Yaskawa INFORM job: DEMO_ROOF_UPPER_0625_3PAINT_5.JBI

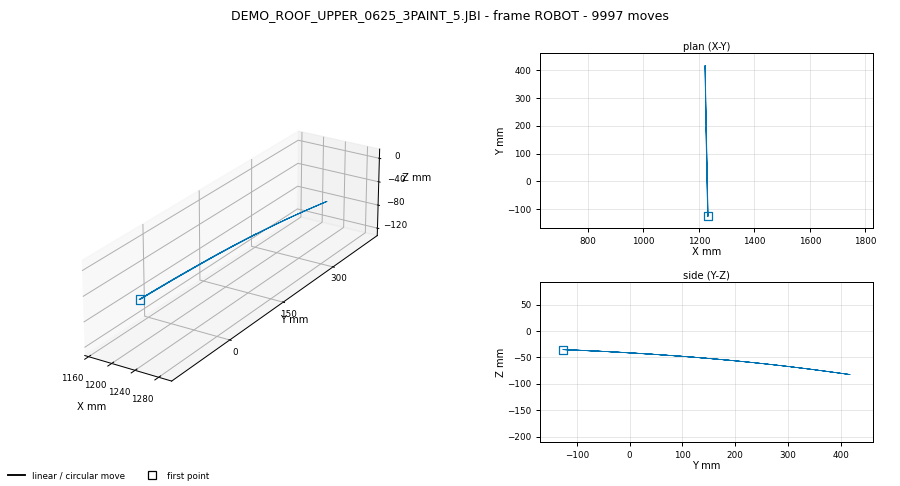
[picture p0: tool path of DEMO_ROOF_UPPER_0625_3PAINT_5.JBI in frame ROBOT, 9997 of 9997 moves have a stored position in this frame; points joined in program order, loops and branches not executed]
/JOB
//NAME DEMO_ROOF_UPPER_0625_3PAINT5
//POS
///NPOS 9997,0,0,0,0,0
///TOOL 0
///USER 0
///POSTYPE ROBOT
///RECTAN
///RCONF 1,0,0,0,0,0,0,0,0,0,0,0,0,0,0,0,0,0,0,0,0,0,0,0
C00000=1233.237,-125.531,-35.008,179.340,5.259,149.111
C00001=1233.231,-125.281,-35.017,179.342,5.259,149.110
C00002=1233.226,-125.032,-35.027,179.345,5.260,149.110
C00003=1233.220,-124.782,-35.037,179.347,5.259,149.109
C00004=1233.215,-124.532,-35.046,179.350,5.260,149.108
C00005=1233.210,-124.282,-35.057,179.352,5.259,149.107
C00006=1233.205,-124.033,-35.067,179.354,5.260,149.107
C00007=1233.199,-123.783,-35.076,179.356,5.260,149.106
C00008=1233.194,-123.533,-35.086,179.359,5.260,149.105
C00009=1233.189,-123.284,-35.096,179.361,5.260,149.105
C00010=1233.184,-123.033,-35.105,179.363,5.259,149.104
C00011=1233.178,-122.784,-35.116,179.366,5.260,149.103
C00012=1233.173,-122.534,-35.125,179.368,5.259,149.103
C00013=1233.168,-122.285,-35.136,179.370,5.260,149.102
C00014=1233.163,-122.034,-35.145,179.372,5.260,149.101
C00015=1233.157,-121.785,-35.155,179.375,5.260,149.101
C00016=1233.152,-121.535,-35.165,179.377,5.260,149.100
C00017=1233.147,-121.286,-35.175,179.379,5.260,149.099
C00018=1233.142,-121.035,-35.185,179.381,5.260,149.099
C00019=1233.136,-120.786,-35.195,179.384,5.260,149.098
C00020=1233.131,-120.536,-35.205,179.386,5.260,149.097
C00021=1233.126,-120.287,-35.215,179.388,5.260,149.096
C00022=1233.121,-120.037,-35.225,179.391,5.260,149.096
C00023=1233.115,-119.787,-35.234,179.393,5.260,149.095
C00024=1233.110,-119.537,-35.244,179.395,5.260,149.094
C00025=1233.105,-119.288,-35.254,179.397,5.260,149.094
C00026=1233.100,-119.038,-35.265,179.400,5.261,149.093
C00027=1233.094,-118.788,-35.275,179.402,5.260,149.092
C00028=1233.089,-118.539,-35.285,179.404,5.260,149.092
C00029=1233.084,-118.288,-35.294,179.407,5.260,149.091
C00030=1233.079,-118.038,-35.304,179.409,5.260,149.090
C00031=1233.073,-117.789,-35.315,179.412,5.260,149.089
C00032=1233.069,-117.539,-35.325,179.414,5.260,149.089
C00033=1233.063,-117.289,-35.335,179.416,5.261,149.088
C00034=1233.058,-117.040,-35.345,179.418,5.260,149.088
C00035=1233.053,-116.791,-35.355,179.421,5.261,149.087
C00036=1233.048,-116.540,-35.365,179.423,5.260,149.086
C00037=1233.042,-116.290,-35.375,179.426,5.261,149.085
C00038=1233.036,-116.041,-35.385,179.428,5.260,149.085
C00039=1233.032,-115.791,-35.395,179.430,5.260,149.084
C00040=1233.026,-115.541,-35.405,179.432,5.261,149.083
C00041=1233.021,-115.292,-35.415,179.435,5.260,149.083
C00042=1233.016,-115.041,-35.426,179.437,5.261,149.082
C00043=1233.011,-114.792,-35.436,179.439,5.260,149.081
C00044=1233.005,-114.543,-35.446,179.441,5.261,149.081
C00045=1233.000,-114.292,-35.456,179.444,5.261,149.080
C00046=1232.995,-114.043,-35.467,179.446,5.261,149.079
C00047=1232.990,-113.794,-35.476,179.448,5.261,149.078
C00048=1232.985,-113.543,-35.487,179.450,5.260,149.078
C00049=1232.979,-113.294,-35.497,179.453,5.261,149.077
C00050=1232.974,-113.044,-35.507,179.455,5.260,149.076
C00051=1232.969,-112.794,-35.518,179.458,5.261,149.076
C00052=1232.964,-112.545,-35.527,179.460,5.260,149.075
C00053=1232.959,-112.295,-35.538,179.463,5.261,149.074
C00054=1232.953,-112.045,-35.548,179.465,5.261,149.073
C00055=1232.948,-111.796,-35.558,179.467,5.261,149.073
C00056=1232.943,-111.545,-35.569,179.470,5.261,149.072
C00057=1232.938,-111.296,-35.579,179.472,5.261,149.072
C00058=1232.932,-111.047,-35.589,179.474,5.261,149.071
C00059=1232.927,-110.796,-35.599,179.476,5.261,149.070
C00060=1232.921,-110.547,-35.610,179.479,5.261,149.069
C00061=1232.916,-110.296,-35.620,179.481,5.261,149.069
C00062=1232.911,-110.047,-35.630,179.483,5.261,149.068
C00063=1232.905,-109.797,-35.641,179.485,5.261,149.067
C00064=1232.901,-109.547,-35.650,179.488,5.261,149.067
C00065=1232.895,-109.298,-35.661,179.490,5.261,149.066
C00066=1232.891,-109.048,-35.672,179.493,5.261,149.065
C00067=1232.885,-108.799,-35.682,179.495,5.261,149.064
C00068=1232.880,-108.549,-35.692,179.498,5.261,149.064
C00069=1232.875,-108.299,-35.703,179.500,5.261,149.063
C00070=1232.869,-108.049,-35.713,179.502,5.261,149.062
C00071=1232.864,-107.799,-35.724,179.504,5.262,149.062
C00072=1232.859,-107.550,-35.733,179.506,5.261,149.061
C00073=1232.854,-107.300,-35.744,179.509,5.262,149.060
C00074=1232.849,-107.051,-35.755,179.511,5.261,149.060
C00075=1232.843,-106.801,-35.765,179.514,5.262,149.059
C00076=1232.838,-106.551,-35.776,179.516,5.261,149.058
C00077=1232.833,-106.301,-35.786,179.518,5.262,149.057
C00078=1232.828,-106.051,-35.796,179.520,5.261,149.057
C00079=1232.822,-105.802,-35.807,179.523,5.262,149.056
C00080=1232.817,-105.552,-35.818,179.525,5.261,149.055
C00081=1232.812,-105.302,-35.828,179.528,5.262,149.055
C00082=1232.807,-105.052,-35.839,179.530,5.262,149.054
C00083=1232.801,-104.803,-35.849,179.533,5.262,149.053
C00084=1232.796,-104.552,-35.859,179.535,5.262,149.052
C00085=1232.792,-104.304,-35.870,179.537,5.261,149.052
C00086=1232.787,-104.054,-35.880,179.540,5.262,149.051
C00087=1232.781,-103.804,-35.891,179.542,5.261,149.050
C00088=1232.776,-103.554,-35.901,179.544,5.262,149.050
C00089=1232.771,-103.305,-35.912,179.546,5.262,149.049
C00090=1232.765,-103.055,-35.922,179.549,5.262,149.048
C00091=1232.760,-102.805,-35.933,179.551,5.262,149.048
C00092=1232.755,-102.556,-35.943,179.553,5.262,149.047
C00093=1232.750,-102.306,-35.954,179.555,5.262,149.046
C00094=1232.745,-102.056,-35.965,179.558,5.262,149.046
C00095=1232.739,-101.806,-35.975,179.560,5.262,149.045
C00096=1232.735,-101.556,-35.986,179.563,5.262,149.044
C00097=1232.729,-101.307,-35.997,179.565,5.262,149.043
C00098=1232.724,-101.057,-36.007,179.568,5.263,149.043
C00099=1232.718,-100.786,-36.019,179.570,5.262,149.042
C00100=1232.712,-100.515,-36.031,179.572,5.263,149.041
C00101=1232.707,-100.244,-36.042,179.575,5.262,149.040
C00102=1232.700,-99.973,-36.053,179.578,5.262,149.040
C00103=1232.696,-99.724,-36.065,179.580,5.262,149.039
C00104=1232.690,-99.474,-36.075,179.582,5.262,149.038
C00105=1232.685,-99.224,-36.086,179.585,5.262,149.037
C00106=1232.680,-98.975,-36.096,179.587,5.263,149.037
C00107=1232.675,-98.725,-36.107,179.589,5.262,149.036
C00108=1232.670,-98.475,-36.118,179.592,5.263,149.035
C00109=1232.665,-98.226,-36.129,179.594,5.262,149.035
C00110=1232.660,-97.975,-36.139,179.597,5.263,149.034
C00111=1232.654,-97.726,-36.150,179.599,5.262,149.033
C00112=1232.649,-97.476,-36.161,179.601,5.263,149.033
C00113=1232.644,-97.227,-36.172,179.603,5.263,149.032
C00114=1232.638,-96.977,-36.183,179.606,5.263,149.031
C00115=1232.633,-96.727,-36.193,179.608,5.263,149.031
C00116=1232.628,-96.477,-36.204,179.611,5.263,149.030
C00117=1232.623,-96.227,-36.215,179.613,5.263,149.029
C00118=1232.618,-95.978,-36.226,179.615,5.263,149.028
C00119=1232.613,-95.728,-36.236,179.617,5.263,149.028
C00120=1232.607,-95.479,-36.247,179.620,5.263,149.027
C00121=1232.602,-95.229,-36.258,179.622,5.263,149.026
C00122=1232.597,-94.979,-36.270,179.624,5.263,149.026
C00123=1232.591,-94.729,-36.280,179.627,5.263,149.025
C00124=1232.587,-94.480,-36.291,179.629,5.263,149.024
C00125=1232.581,-94.230,-36.301,179.632,5.263,149.023
C00126=1232.576,-93.981,-36.313,179.634,5.263,149.023
C00127=1232.571,-93.730,-36.323,179.637,5.263,149.022
C00128=1232.565,-93.481,-36.335,179.639,5.263,149.021
C00129=1232.560,-93.231,-36.345,179.641,5.264,149.021
C00130=1232.555,-92.982,-36.356,179.643,5.263,149.020
C00131=1232.550,-92.732,-36.367,179.646,5.264,149.019
C00132=1232.545,-92.482,-36.378,179.648,5.263,149.018
C00133=1232.539,-92.232,-36.389,179.651,5.264,149.018
C00134=1232.534,-91.983,-36.400,179.653,5.263,149.017
C00135=1232.529,-91.732,-36.411,179.656,5.264,149.016
C00136=1232.524,-91.483,-36.422,179.658,5.263,149.016
C00137=1232.519,-91.234,-36.433,179.660,5.264,149.015
C00138=1232.514,-90.983,-36.444,179.662,5.264,149.014
C00139=1232.508,-90.734,-36.455,179.665,5.264,149.013
C00140=1232.503,-90.484,-36.466,179.667,5.264,149.013
C00141=1232.499,-90.234,-36.477,179.670,5.264,149.012
C00142=1232.493,-89.985,-36.489,179.672,5.264,149.011
C00143=1232.488,-89.735,-36.499,179.675,5.264,149.011
C00144=1232.482,-89.486,-36.510,179.677,5.264,149.010
C00145=1232.477,-89.236,-36.521,179.679,5.264,149.009
C00146=1232.472,-88.986,-36.532,179.682,5.264,149.008
C00147=1232.467,-88.736,-36.544,179.684,5.264,149.008
C00148=1232.462,-88.487,-36.554,179.686,5.264,149.007
C00149=1232.457,-88.237,-36.565,179.688,5.264,149.006
C00150=1232.451,-87.987,-36.577,179.691,5.264,149.006
C00151=1232.446,-87.738,-36.587,179.693,5.264,149.005
C00152=1232.441,-87.488,-36.599,179.696,5.264,149.004
C00153=1232.436,-87.238,-36.611,179.698,5.264,149.004
C00154=1232.430,-86.989,-36.621,179.701,5.264,149.003
C00155=1232.425,-86.739,-36.632,179.703,5.264,149.002
C00156=1232.421,-86.489,-36.643,179.705,5.264,149.001
C00157=1232.415,-86.239,-36.655,179.707,5.264,149.001
C00158=1232.410,-85.990,-36.665,179.710,5.265,149.000
C00159=1232.405,-85.740,-36.677,179.712,5.264,148.999
C00160=1232.400,-85.490,-36.689,179.715,5.265,148.999
C00161=1232.394,-85.241,-36.700,179.717,5.264,148.998
C00162=1232.389,-84.991,-36.710,179.720,5.265,148.997
C00163=1232.384,-84.741,-36.722,179.722,5.264,148.996
C00164=1232.379,-84.491,-36.733,179.724,5.265,148.996
C00165=1232.374,-84.243,-36.744,179.726,5.265,148.995
C00166=1232.368,-83.992,-36.755,179.729,5.265,148.994
C00167=1232.363,-83.742,-36.767,179.731,5.265,148.994
C00168=1232.359,-83.493,-36.778,179.733,5.266,148.993
C00169=1232.353,-83.243,-36.789,179.736,5.265,148.992
C00170=1232.348,-82.994,-36.801,179.738,5.266,148.992
C00171=1232.342,-82.743,-36.812,179.740,5.265,148.991
C00172=1232.338,-82.494,-36.823,179.743,5.266,148.990
C00173=1232.332,-82.245,-36.834,179.745,5.265,148.990
C00174=1232.327,-81.995,-36.846,179.748,5.266,148.989
C00175=1232.322,-81.745,-36.857,179.750,5.265,148.988
C00176=1232.317,-81.495,-36.869,179.753,5.266,148.987
C00177=1232.312,-81.246,-36.880,179.755,5.265,148.986
C00178=1232.306,-80.996,-36.891,179.758,5.266,148.986
C00179=1232.301,-80.746,-36.903,179.760,5.265,148.985
C00180=1232.296,-80.497,-36.914,179.763,5.266,148.984
C00181=1232.291,-80.247,-36.926,179.765,5.265,148.984
C00182=1232.286,-79.998,-36.937,179.767,5.266,148.983
C00183=1232.280,-79.748,-36.949,179.769,5.266,148.982
C00184=1232.276,-79.498,-36.960,179.772,5.266,148.981
C00185=1232.271,-79.248,-36.971,179.774,5.266,148.981
C00186=1232.265,-78.999,-36.983,179.777,5.266,148.980
C00187=1232.260,-78.749,-36.993,179.779,5.266,148.979
C00188=1232.254,-78.499,-37.005,179.782,5.266,148.979
C00189=1232.250,-78.249,-37.016,179.784,5.266,148.978
C00190=1232.244,-77.999,-37.028,179.786,5.266,148.977
C00191=1232.240,-77.750,-37.040,179.788,5.266,148.977
C00192=1232.234,-77.500,-37.051,179.791,5.266,148.976
C00193=1232.229,-77.251,-37.062,179.793,5.266,148.975
C00194=1232.223,-77.001,-37.074,179.796,5.267,148.974
C00195=1232.219,-76.751,-37.086,179.798,5.266,148.974
C00196=1232.213,-76.502,-37.097,179.801,5.267,148.973
C00197=1232.209,-76.252,-37.109,179.803,5.266,148.972
C00198=1232.203,-76.002,-37.121,179.805,5.267,148.972
C00199=1232.198,-75.753,-37.132,179.807,5.267,148.971
C00200=1232.192,-75.503,-37.143,179.810,5.267,148.970
C00201=1232.187,-75.253,-37.155,179.812,5.267,148.969
C00202=1232.182,-75.004,-37.167,179.815,5.267,148.969
C00203=1232.177,-74.733,-37.180,179.818,5.268,148.968
C00204=1232.171,-74.463,-37.191,179.820,5.267,148.967
C00205=1232.165,-74.193,-37.204,179.822,5.268,148.967
C00206=1232.160,-73.922,-37.217,179.825,5.268,148.966
C00207=1232.155,-73.673,-37.228,179.828,5.267,148.965
C00208=1232.149,-73.423,-37.240,179.830,5.268,148.964
C00209=1232.144,-73.173,-37.252,179.832,5.268,148.964
C00210=1232.139,-72.924,-37.263,179.835,5.268,148.963
C00211=1232.134,-72.674,-37.275,179.837,5.268,148.962
C00212=1232.129,-72.424,-37.287,179.840,5.268,148.961
C00213=1232.124,-72.174,-37.298,179.842,5.268,148.961
C00214=1232.119,-71.925,-37.311,179.845,5.268,148.960
C00215=1232.114,-71.675,-37.322,179.847,5.268,148.959
C00216=1232.108,-71.426,-37.334,179.849,5.268,148.959
C00217=1232.103,-71.176,-37.345,179.851,5.268,148.958
C00218=1232.098,-70.927,-37.357,179.854,5.269,148.957
C00219=1232.092,-70.677,-37.369,179.856,5.268,148.956
C00220=1232.088,-70.427,-37.380,179.859,5.269,148.956
C00221=1232.083,-70.178,-37.393,179.861,5.268,148.955
C00222=1232.077,-69.928,-37.405,179.864,5.269,148.954
C00223=1232.072,-69.678,-37.416,179.866,5.268,148.954
C00224=1232.067,-69.428,-37.428,179.868,5.269,148.953
C00225=1232.062,-69.178,-37.440,179.870,5.269,148.952
C00226=1232.057,-68.929,-37.451,179.873,5.269,148.952
C00227=1232.052,-68.679,-37.464,179.875,5.269,148.951
C00228=1232.046,-68.429,-37.476,179.878,5.269,148.950
C00229=1232.042,-68.180,-37.487,179.880,5.269,148.949
C00230=1232.036,-67.930,-37.498,179.883,5.269,148.949
C00231=1232.030,-67.681,-37.511,179.885,5.270,148.948
C00232=1232.026,-67.432,-37.522,179.887,5.269,148.947
C00233=1232.020,-67.182,-37.534,179.890,5.270,148.947
C00234=1232.015,-66.932,-37.546,179.892,5.270,148.946
C00235=1232.010,-66.682,-37.559,179.895,5.270,148.945
C00236=1232.005,-66.433,-37.570,179.897,5.270,148.944
C00237=1232.000,-66.183,-37.582,179.900,5.270,148.944
C00238=1231.994,-65.933,-37.594,179.902,5.270,148.943
C00239=1231.990,-65.684,-37.606,179.904,5.270,148.942
C00240=1231.984,-65.434,-37.618,179.906,5.270,148.942
C00241=1231.979,-65.184,-37.629,179.910,5.270,148.941
C00242=1231.974,-64.935,-37.642,179.912,5.270,148.940
C00243=1231.969,-64.685,-37.653,179.914,5.270,148.939
C00244=1231.964,-64.435,-37.665,179.916,5.270,148.939
C00245=1231.959,-64.186,-37.678,179.919,5.270,148.938
C00246=1231.953,-63.936,-37.690,179.921,5.270,148.937
C00247=1231.949,-63.686,-37.701,179.924,5.271,148.936
C00248=1231.943,-63.437,-37.714,179.927,5.271,148.936
C00249=1231.938,-63.187,-37.725,179.929,5.271,148.935
C00250=1231.933,-62.937,-37.737,179.931,5.271,148.934
C00251=1231.927,-62.688,-37.750,179.933,5.271,148.934
C00252=1231.923,-62.438,-37.761,179.936,5.271,148.933
C00253=1231.918,-62.189,-37.774,179.938,5.271,148.932
C00254=1231.912,-61.939,-37.786,179.941,5.271,148.932
C00255=1231.907,-61.689,-37.798,179.943,5.271,148.931
C00256=1231.902,-61.439,-37.811,179.946,5.272,148.930
C00257=1231.898,-61.189,-37.822,179.948,5.271,148.929
C00258=1231.892,-60.940,-37.834,179.950,5.272,148.929
C00259=1231.887,-60.690,-37.846,179.952,5.271,148.928
C00260=1231.882,-60.440,-37.858,179.955,5.272,148.927
C00261=1231.876,-60.191,-37.871,179.958,5.272,148.927
C00262=1231.871,-59.941,-37.883,179.960,5.272,148.926
C00263=1231.867,-59.692,-37.895,179.962,5.272,148.925
C00264=1231.861,-59.442,-37.907,179.965,5.272,148.924
C00265=1231.856,-59.193,-37.919,179.967,5.273,148.924
C00266=1231.851,-58.943,-37.931,179.969,5.272,148.923
C00267=1231.846,-58.693,-37.944,179.972,5.273,148.922
C00268=1231.840,-58.443,-37.956,179.974,5.272,148.922
C00269=1231.835,-58.194,-37.968,179.977,5.273,148.921
C00270=1231.831,-57.944,-37.980,179.979,5.273,148.920
C00271=1231.826,-57.694,-37.992,179.981,5.273,148.920
C00272=1231.820,-57.444,-38.004,179.984,5.274,148.919
C00273=1231.815,-57.195,-38.017,179.987,5.273,148.918
C00274=1231.810,-56.945,-38.029,179.989,5.273,148.917
C00275=1231.805,-56.696,-38.041,179.991,5.273,148.916
C00276=1231.800,-56.447,-38.054,179.994,5.273,148.916
C00277=1231.794,-56.197,-38.066,179.996,5.273,148.915
C00278=1231.789,-55.947,-38.078,179.999,5.274,148.914
C00279=1231.784,-55.697,-38.091,-179.999,5.273,148.914
C00280=1231.779,-55.447,-38.103,-179.996,5.274,148.913
C00281=1231.774,-55.198,-38.115,-179.994,5.274,148.912
C00282=1231.769,-54.948,-38.127,-179.992,5.274,148.912
C00283=1231.764,-54.699,-38.140,-179.989,5.274,148.911
C00284=1231.759,-54.449,-38.152,-179.987,5.274,148.910
C00285=1231.754,-54.200,-38.164,-179.984,5.275,148.909
C00286=1231.749,-53.950,-38.177,-179.982,5.274,148.909
C00287=1231.744,-53.700,-38.189,-179.979,5.275,148.908
C00288=1231.738,-53.451,-38.202,-179.977,5.274,148.907
C00289=1231.733,-53.201,-38.214,-179.975,5.275,148.907
C00290=1231.728,-52.951,-38.226,-179.972,5.275,148.906
C00291=1231.723,-52.702,-38.239,-179.970,5.275,148.905
C00292=1231.718,-52.451,-38.251,-179.967,5.276,148.904
C00293=1231.713,-52.202,-38.264,-179.965,5.275,148.904
C00294=1231.708,-51.953,-38.276,-179.962,5.276,148.903
C00295=1231.703,-51.703,-38.289,-179.960,5.275,148.902
C00296=1231.697,-51.453,-38.301,-179.958,5.276,148.902
C00297=1231.692,-51.204,-38.313,-179.955,5.276,148.901
C00298=1231.687,-50.954,-38.326,-179.953,5.276,148.900
C00299=1231.682,-50.704,-38.338,-179.950,5.276,148.899
C00300=1231.677,-50.455,-38.351,-179.948,5.276,148.899
C00301=1231.672,-50.206,-38.363,-179.945,5.276,148.898
C00302=1231.667,-49.956,-38.376,-179.943,5.276,148.897
C00303=1231.662,-49.706,-38.388,-179.940,5.276,148.897
C00304=1231.657,-49.456,-38.401,-179.938,5.276,148.896
C00305=1231.651,-49.207,-38.414,-179.936,5.277,148.895
C00306=1231.646,-48.957,-38.427,-179.933,5.277,148.894
C00307=1231.640,-48.687,-38.440,-179.931,5.277,148.894
C00308=1231.635,-48.417,-38.453,-179.928,5.277,148.893
C00309=1231.629,-48.148,-38.467,-179.925,5.277,148.892
C00310=1231.624,-47.878,-38.481,-179.923,5.277,148.891
C00311=1231.619,-47.628,-38.493,-179.920,5.278,148.891
C00312=1231.614,-47.379,-38.505,-179.918,5.278,148.890
C00313=1231.609,-47.129,-38.518,-179.915,5.278,148.889
C00314=1231.604,-46.880,-38.531,-179.913,5.278,148.889
C00315=1231.598,-46.630,-38.544,-179.911,5.278,148.888
C00316=1231.593,-46.381,-38.557,-179.908,5.278,148.887
C00317=1231.588,-46.131,-38.570,-179.906,5.278,148.886
C00318=1231.583,-45.881,-38.582,-179.903,5.279,148.886
C00319=1231.578,-45.631,-38.594,-179.901,5.279,148.885
C00320=1231.573,-45.382,-38.607,-179.899,5.279,148.884
C00321=1231.568,-45.132,-38.620,-179.896,5.279,148.884
C00322=1231.562,-44.882,-38.633,-179.894,5.279,148.883
C00323=1231.557,-44.633,-38.646,-179.891,5.279,148.882
C00324=1231.552,-44.384,-38.658,-179.889,5.279,148.881
C00325=1231.548,-44.134,-38.671,-179.886,5.279,148.881
C00326=1231.542,-43.884,-38.684,-179.883,5.280,148.880
C00327=1231.537,-43.634,-38.696,-179.881,5.279,148.879
C00328=1231.532,-43.384,-38.709,-179.878,5.280,148.879
C00329=1231.527,-43.135,-38.722,-179.876,5.279,148.878
C00330=1231.521,-42.886,-38.734,-179.874,5.280,148.877
C00331=1231.516,-42.636,-38.747,-179.871,5.280,148.876
C00332=1231.512,-42.386,-38.760,-179.869,5.280,148.876
C00333=1231.506,-42.137,-38.773,-179.866,5.281,148.875
C00334=1231.501,-41.887,-38.786,-179.864,5.280,148.874
C00335=1231.496,-41.637,-38.799,-179.862,5.281,148.874
C00336=1231.491,-41.388,-38.811,-179.859,5.281,148.873
C00337=1231.485,-41.138,-38.825,-179.857,5.281,148.872
C00338=1231.481,-40.888,-38.838,-179.854,5.281,148.871
C00339=1231.476,-40.639,-38.850,-179.852,5.281,148.871
C00340=1231.471,-40.390,-38.863,-179.849,5.282,148.870
C00341=1231.466,-40.140,-38.876,-179.847,5.281,148.869
C00342=1231.460,-39.890,-38.889,-179.845,5.282,148.869
C00343=1231.455,-39.641,-38.901,-179.842,5.282,148.868
C00344=1231.451,-39.391,-38.914,-179.840,5.282,148.867
C00345=1231.445,-39.141,-38.928,-179.837,5.283,148.867
C00346=1231.440,-38.892,-38.940,-179.835,5.282,148.866
C00347=1231.435,-38.642,-38.953,-179.832,5.282,148.865
C00348=1231.430,-38.393,-38.967,-179.829,5.283,148.864
C00349=1231.425,-38.143,-38.980,-179.827,5.282,148.864
C00350=1231.420,-37.893,-38.993,-179.825,5.283,148.863
C00351=1231.415,-37.644,-39.005,-179.823,5.283,148.862
C00352=1231.409,-37.394,-39.019,-179.820,5.283,148.861
C00353=1231.404,-37.144,-39.031,-179.817,5.284,148.861
C00354=1231.399,-36.895,-39.044,-179.815,5.283,148.860
C00355=1231.394,-36.645,-39.058,-179.812,5.284,148.859
C00356=1231.389,-36.395,-39.070,-179.810,5.284,148.859
C00357=1231.384,-36.147,-39.084,-179.808,5.284,148.858
C00358=1231.379,-35.896,-39.097,-179.805,5.285,148.857
C00359=1231.374,-35.647,-39.110,-179.803,5.284,148.857
C00360=1231.369,-35.397,-39.123,-179.800,5.285,148.856
C00361=1231.363,-35.147,-39.136,-179.798,5.284,148.855
C00362=1231.358,-34.898,-39.148,-179.796,5.285,148.854
C00363=1231.353,-34.648,-39.163,-179.793,5.285,148.854
C00364=1231.348,-34.399,-39.175,-179.791,5.285,148.853
C00365=1231.344,-34.149,-39.188,-179.788,5.286,148.852
C00366=1231.338,-33.899,-39.202,-179.786,5.285,148.852
C00367=1231.333,-33.649,-39.214,-179.783,5.286,148.851
C00368=1231.328,-33.401,-39.228,-179.781,5.286,148.850
C00369=1231.322,-33.151,-39.241,-179.779,5.286,148.850
C00370=1231.318,-32.901,-39.254,-179.775,5.286,148.849
C00371=1231.312,-32.651,-39.267,-179.773,5.287,148.848
C00372=1231.308,-32.402,-39.281,-179.771,5.286,148.847
C00373=1231.302,-32.152,-39.294,-179.768,5.287,148.847
C00374=1231.297,-31.902,-39.307,-179.766,5.286,148.846
C00375=1231.292,-31.653,-39.320,-179.763,5.287,148.845
C00376=1231.287,-31.403,-39.334,-179.761,5.287,148.844
C00377=1231.282,-31.154,-39.346,-179.759,5.287,148.844
C00378=1231.276,-30.904,-39.360,-179.756,5.288,148.843
C00379=1231.272,-30.655,-39.373,-179.754,5.287,148.842
C00380=1231.266,-30.405,-39.387,-179.751,5.288,148.842
C00381=1231.262,-30.155,-39.400,-179.749,5.288,148.841
C00382=1231.256,-29.906,-39.413,-179.746,5.288,148.840
C00383=1231.252,-29.656,-39.426,-179.744,5.289,148.840
C00384=1231.246,-29.407,-39.440,-179.741,5.289,148.839
C00385=1231.242,-29.157,-39.453,-179.739,5.289,148.838
C00386=1231.237,-28.908,-39.466,-179.736,5.289,148.837
C00387=1231.231,-28.658,-39.479,-179.734,5.289,148.837
C00388=1231.226,-28.409,-39.493,-179.732,5.289,148.836
C00389=1231.221,-28.159,-39.506,-179.729,5.290,148.835
C00390=1231.216,-27.909,-39.519,-179.727,5.290,148.835
C00391=1231.211,-27.660,-39.533,-179.724,5.290,148.834
C00392=1231.205,-27.410,-39.546,-179.722,5.291,148.833
C00393=1231.201,-27.161,-39.560,-179.719,5.290,148.832
C00394=1231.195,-26.911,-39.573,-179.716,5.290,148.832
C00395=1231.191,-26.662,-39.587,-179.714,5.290,148.831
C00396=1231.185,-26.412,-39.600,-179.712,5.291,148.830
C00397=1231.181,-26.162,-39.613,-179.709,5.291,148.830
C00398=1231.175,-25.913,-39.627,-179.707,5.291,148.829
C00399=1231.170,-25.663,-39.640,-179.704,5.291,148.828
C00400=1231.166,-25.413,-39.654,-179.702,5.292,148.827
C00401=1231.160,-25.164,-39.667,-179.699,5.292,148.827
C00402=1231.155,-24.914,-39.681,-179.697,5.292,148.826
C00403=1231.150,-24.664,-39.694,-179.694,5.293,148.825
C00404=1231.145,-24.415,-39.708,-179.692,5.292,148.825
C00405=1231.139,-24.165,-39.721,-179.689,5.293,148.824
C00406=1231.135,-23.916,-39.735,-179.687,5.292,148.823
C00407=1231.129,-23.666,-39.748,-179.685,5.293,148.823
C00408=1231.124,-23.417,-39.762,-179.682,5.294,148.822
C00409=1231.120,-23.167,-39.775,-179.680,5.293,148.821
C00410=1231.114,-22.918,-39.789,-179.677,5.294,148.821
C00411=1231.109,-22.648,-39.804,-179.675,5.294,148.820
C00412=1231.104,-22.379,-39.818,-179.671,5.294,148.819
C00413=1231.098,-22.110,-39.833,-179.669,5.294,148.818
C00414=1231.092,-21.840,-39.848,-179.667,5.295,148.817
C00415=1231.088,-21.591,-39.862,-179.664,5.295,148.817
C00416=1231.082,-21.341,-39.874,-179.662,5.295,148.816
C00417=1231.077,-21.092,-39.889,-179.659,5.295,148.815
C00418=1231.072,-20.842,-39.903,-179.657,5.296,148.815
C00419=1231.067,-20.593,-39.916,-179.655,5.295,148.814
C00420=1231.062,-20.343,-39.930,-179.651,5.296,148.813
C00421=1231.057,-20.093,-39.943,-179.649,5.296,148.812
C00422=1231.052,-19.844,-39.957,-179.647,5.296,148.812
C00423=1231.047,-19.594,-39.971,-179.644,5.296,148.811
C00424=1231.042,-19.345,-39.984,-179.641,5.297,148.810
C00425=1231.037,-19.095,-39.998,-179.639,5.297,148.810
C00426=1231.032,-18.845,-40.012,-179.637,5.297,148.809
C00427=1231.026,-18.596,-40.025,-179.634,5.298,148.808
C00428=1231.022,-18.346,-40.039,-179.632,5.297,148.808
C00429=1231.017,-18.097,-40.053,-179.629,5.298,148.807
C00430=1231.011,-17.847,-40.067,-179.627,5.298,148.806
C00431=1231.006,-17.597,-40.081,-179.624,5.298,148.805
C00432=1231.002,-17.349,-40.094,-179.622,5.299,148.805
C00433=1230.996,-17.098,-40.108,-179.619,5.299,148.804
C00434=1230.991,-16.849,-40.122,-179.617,5.299,148.803
C00435=1230.986,-16.600,-40.136,-179.614,5.299,148.803
C00436=1230.982,-16.350,-40.150,-179.612,5.299,148.802
C00437=1230.976,-16.100,-40.163,-179.610,5.299,148.801
C00438=1230.971,-15.851,-40.177,-179.607,5.300,148.801
C00439=1230.966,-15.601,-40.191,-179.605,5.300,148.800
C00440=1230.961,-15.351,-40.206,-179.602,5.300,148.799
C00441=1230.956,-15.102,-40.218,-179.600,5.301,148.799
C00442=1230.951,-14.852,-40.232,-179.598,5.300,148.798
C00443=1230.946,-14.603,-40.247,-179.595,5.301,148.797
C00444=1230.940,-14.354,-40.261,-179.592,5.301,148.796
C00445=1230.935,-14.104,-40.275,-179.590,5.301,148.796
C00446=1230.931,-13.854,-40.288,-179.587,5.302,148.795
C00447=1230.926,-13.604,-40.302,-179.585,5.302,148.794
C00448=1230.920,-13.355,-40.316,-179.583,5.302,148.794
C00449=1230.915,-13.106,-40.330,-179.580,5.302,148.793
C00450=1230.910,-12.856,-40.345,-179.577,5.303,148.792
C00451=1230.906,-12.607,-40.358,-179.574,5.303,148.791
C00452=1230.900,-12.357,-40.371,-179.572,5.303,148.791
C00453=1230.895,-12.107,-40.386,-179.570,5.303,148.790
C00454=1230.890,-11.857,-40.400,-179.567,5.304,148.789
C00455=1230.885,-11.608,-40.414,-179.565,5.304,148.789
C00456=1230.880,-11.359,-40.428,-179.562,5.304,148.788
C00457=1230.875,-11.109,-40.443,-179.559,5.305,148.787
C00458=1230.871,-10.860,-40.456,-179.557,5.304,148.786
C00459=1230.865,-10.611,-40.470,-179.555,5.305,148.786
C00460=1230.860,-10.360,-40.484,-179.552,5.305,148.785
C00461=1230.855,-10.111,-40.498,-179.550,5.305,148.784
C00462=1230.850,-9.861,-40.512,-179.547,5.306,148.784
C00463=1230.845,-9.612,-40.526,-179.545,5.306,148.783
C00464=1230.840,-9.362,-40.540,-179.543,5.306,148.782
C00465=1230.835,-9.112,-40.555,-179.540,5.306,148.782
C00466=1230.830,-8.863,-40.569,-179.537,5.307,148.781
C00467=1230.824,-8.614,-40.583,-179.535,5.306,148.780
C00468=1230.820,-8.364,-40.597,-179.533,5.307,148.780
C00469=1230.815,-8.115,-40.611,-179.530,5.308,148.779
C00470=1230.810,-7.865,-40.625,-179.528,5.307,148.778
C00471=1230.805,-7.615,-40.639,-179.525,5.308,148.777
C00472=1230.799,-7.366,-40.653,-179.523,5.308,148.777
C00473=1230.795,-7.116,-40.668,-179.520,5.309,148.776
C00474=1230.790,-6.867,-40.682,-179.518,5.309,148.775
C00475=1230.785,-6.617,-40.696,-179.515,5.309,148.775
C00476=1230.780,-6.367,-40.710,-179.512,5.310,148.774
C00477=1230.774,-6.118,-40.724,-179.510,5.309,148.773
C00478=1230.769,-5.869,-40.739,-179.508,5.310,148.773
C00479=1230.764,-5.619,-40.753,-179.505,5.310,148.772
C00480=1230.759,-5.369,-40.767,-179.503,5.310,148.771
C00481=1230.754,-5.119,-40.781,-179.500,5.311,148.771
C00482=1230.750,-4.870,-40.796,-179.498,5.311,148.770
C00483=1230.744,-4.621,-40.810,-179.496,5.311,148.769
C00484=1230.739,-4.372,-40.825,-179.493,5.311,148.769
C00485=1230.734,-4.122,-40.839,-179.490,5.312,148.768
C00486=1230.729,-3.872,-40.853,-179.488,5.312,148.767
C00487=1230.724,-3.622,-40.867,-179.486,5.312,148.766
C00488=1230.719,-3.373,-40.882,-179.482,5.312,148.766
C00489=1230.714,-3.124,-40.896,-179.480,5.313,148.765
C00490=1230.709,-2.875,-40.911,-179.478,5.312,148.764
C00491=1230.704,-2.625,-40.925,-179.475,5.313,148.763
C00492=1230.699,-2.375,-40.939,-179.472,5.313,148.763
C00493=1230.694,-2.126,-40.953,-179.470,5.314,148.762
C00494=1230.689,-1.876,-40.968,-179.468,5.314,148.761
C00495=1230.684,-1.626,-40.983,-179.465,5.314,148.761
C00496=1230.679,-1.377,-40.998,-179.462,5.315,148.760
C00497=1230.673,-1.128,-41.012,-179.460,5.315,148.759
C00498=1230.668,-0.878,-41.026,-179.458,5.315,148.759
C00499=1230.663,-0.628,-41.040,-179.455,5.316,148.758
C00500=1230.659,-0.379,-41.054,-179.452,5.316,148.757
C00501=1230.654,-0.130,-41.069,-179.450,5.316,148.757
C00502=1230.649,0.120,-41.084,-179.448,5.316,148.756
C00503=1230.644,0.370,-41.098,-179.445,5.317,148.755
C00504=1230.638,0.620,-41.113,-179.443,5.317,148.754
C00505=1230.634,0.869,-41.128,-179.440,5.317,148.754
C00506=1230.629,1.119,-41.142,-179.438,5.318,148.753
C00507=1230.623,1.368,-41.156,-179.435,5.318,148.752
C00508=1230.618,1.617,-41.170,-179.433,5.318,148.752
C00509=1230.613,1.867,-41.185,-179.430,5.318,148.751
C00510=1230.609,2.116,-41.199,-179.428,5.319,148.750
C00511=1230.603,2.366,-41.214,-179.425,5.319,148.750
C00512=1230.598,2.615,-41.229,-179.423,5.319,148.749
C00513=1230.593,2.865,-41.244,-179.420,5.320,148.748
C00514=1230.588,3.115,-41.258,-179.417,5.320,148.748
C00515=1230.583,3.384,-41.274,-179.415,5.320,148.747
C00516=1230.577,3.653,-41.290,-179.413,5.320,148.746
C00517=1230.572,3.921,-41.306,-179.410,5.321,148.745
C00518=1230.567,4.190,-41.321,-179.407,5.321,148.745
C00519=1230.562,4.440,-41.336,-179.404,5.322,148.744
C00520=1230.557,4.689,-41.351,-179.402,5.322,148.743
C00521=1230.552,4.939,-41.365,-179.400,5.322,148.743
C00522=1230.547,5.189,-41.380,-179.397,5.322,148.742
C00523=1230.542,5.437,-41.394,-179.394,5.323,148.741
C00524=1230.536,5.687,-41.409,-179.392,5.323,148.740
C00525=1230.531,5.936,-41.424,-179.390,5.323,148.740
C00526=1230.526,6.186,-41.439,-179.387,5.324,148.739
C00527=1230.521,6.436,-41.453,-179.384,5.324,148.738
C00528=1230.516,6.685,-41.468,-179.382,5.324,148.738
C00529=1230.511,6.935,-41.483,-179.380,5.325,148.737
C00530=1230.506,7.184,-41.498,-179.377,5.325,148.736
C00531=1230.501,7.434,-41.512,-179.374,5.326,148.736
C00532=1230.496,7.683,-41.528,-179.372,5.325,148.735
C00533=1230.491,7.933,-41.542,-179.369,5.326,148.734
C00534=1230.487,8.183,-41.557,-179.367,5.326,148.734
C00535=1230.481,8.433,-41.572,-179.364,5.327,148.733
C00536=1230.477,8.682,-41.587,-179.362,5.327,148.732
C00537=1230.472,8.931,-41.601,-179.359,5.327,148.732
C00538=1230.467,9.180,-41.616,-179.357,5.328,148.731
C00539=1230.461,9.430,-41.631,-179.354,5.328,148.730
C00540=1230.457,9.680,-41.646,-179.352,5.328,148.730
C00541=1230.452,9.929,-41.660,-179.349,5.329,148.729
C00542=1230.446,10.179,-41.676,-179.347,5.329,148.728
C00543=1230.441,10.428,-41.690,-179.344,5.330,148.727
C00544=1230.437,10.677,-41.705,-179.342,5.329,148.727
C00545=1230.431,10.927,-41.721,-179.339,5.330,148.726
C00546=1230.426,11.177,-41.735,-179.337,5.330,148.725
C00547=1230.422,11.426,-41.750,-179.334,5.331,148.725
C00548=1230.416,11.676,-41.765,-179.332,5.331,148.724
C00549=1230.411,11.925,-41.780,-179.329,5.331,148.723
C00550=1230.406,12.174,-41.796,-179.327,5.332,148.723
C00551=1230.401,12.424,-41.810,-179.324,5.332,148.722
C00552=1230.396,12.673,-41.825,-179.322,5.332,148.721
C00553=1230.391,12.923,-41.840,-179.319,5.333,148.721
C00554=1230.387,13.173,-41.855,-179.317,5.333,148.720
C00555=1230.381,13.422,-41.871,-179.314,5.334,148.719
C00556=1230.376,13.672,-41.885,-179.311,5.334,148.719
C00557=1230.372,13.921,-41.900,-179.309,5.334,148.718
C00558=1230.366,14.170,-41.916,-179.307,5.334,148.717
C00559=1230.361,14.420,-41.930,-179.304,5.335,148.716
C00560=1230.356,14.670,-41.945,-179.301,5.336,148.716
C00561=1230.351,14.919,-41.960,-179.299,5.335,148.715
C00562=1230.346,15.168,-41.976,-179.297,5.336,148.714
C00563=1230.342,15.418,-41.991,-179.294,5.336,148.714
C00564=1230.336,15.668,-42.006,-179.291,5.337,148.713
C00565=1230.332,15.917,-42.021,-179.289,5.337,148.712
C00566=1230.327,16.167,-42.035,-179.287,5.337,148.712
C00567=1230.321,16.416,-42.051,-179.284,5.338,148.711
C00568=1230.317,16.665,-42.066,-179.281,5.338,148.710
C00569=1230.311,16.915,-42.082,-179.279,5.339,148.710
C00570=1230.306,17.164,-42.096,-179.277,5.338,148.709
C00571=1230.301,17.414,-42.112,-179.274,5.339,148.708
C00572=1230.297,17.663,-42.127,-179.271,5.340,148.708
C00573=1230.291,17.913,-42.142,-179.269,5.340,148.707
C00574=1230.287,18.162,-42.157,-179.267,5.340,148.706
C00575=1230.281,18.412,-42.172,-179.264,5.341,148.706
C00576=1230.276,18.661,-42.187,-179.262,5.341,148.705
C00577=1230.272,18.911,-42.203,-179.259,5.342,148.704
C00578=1230.266,19.161,-42.219,-179.257,5.342,148.704
C00579=1230.262,19.410,-42.234,-179.254,5.342,148.703
C00580=1230.256,19.659,-42.249,-179.252,5.343,148.702
C00581=1230.251,19.909,-42.264,-179.249,5.343,148.702
C00582=1230.246,20.159,-42.280,-179.247,5.344,148.701
C00583=1230.242,20.408,-42.295,-179.244,5.344,148.700
C00584=1230.236,20.657,-42.310,-179.242,5.344,148.700
C00585=1230.232,20.906,-42.325,-179.239,5.345,148.699
C00586=1230.226,21.156,-42.341,-179.236,5.345,148.698
C00587=1230.222,21.406,-42.357,-179.234,5.346,148.698
C00588=1230.217,21.655,-42.372,-179.231,5.346,148.697
C00589=1230.212,21.904,-42.387,-179.229,5.346,148.696
C00590=1230.207,22.154,-42.402,-179.226,5.346,148.696
C00591=1230.201,22.404,-42.417,-179.224,5.347,148.695
C00592=1230.196,22.654,-42.433,-179.221,5.348,148.694
C00593=1230.192,22.903,-42.448,-179.219,5.348,148.694
C00594=1230.186,23.152,-42.464,-179.216,5.348,148.693
C00595=1230.182,23.401,-42.479,-179.214,5.348,148.692
C00596=1230.177,23.651,-42.495,-179.211,5.349,148.691
C00597=1230.172,23.901,-42.510,-179.209,5.349,148.691
C00598=1230.167,24.150,-42.525,-179.206,5.350,148.690
C00599=1230.162,24.399,-42.541,-179.204,5.350,148.689
C00600=1230.157,24.649,-42.557,-179.201,5.350,148.689
C00601=1230.152,24.898,-42.572,-179.199,5.351,148.688
C00602=1230.147,25.148,-42.587,-179.196,5.351,148.687
C00603=1230.141,25.397,-42.603,-179.193,5.352,148.687
C00604=1230.137,25.647,-42.618,-179.191,5.352,148.686
C00605=1230.132,25.896,-42.634,-179.189,5.352,148.685
C00606=1230.126,26.146,-42.650,-179.186,5.353,148.685
C00607=1230.122,26.394,-42.665,-179.183,5.353,148.684
C00608=1230.117,26.644,-42.681,-179.181,5.354,148.684
C00609=1230.112,26.894,-42.697,-179.179,5.354,148.683
C00610=1230.107,27.143,-42.712,-179.176,5.355,148.682
C00611=1230.103,27.393,-42.728,-179.174,5.355,148.681
C00612=1230.097,27.642,-42.743,-179.171,5.356,148.681
C00613=1230.092,27.892,-42.759,-179.168,5.356,148.680
C00614=1230.087,28.142,-42.775,-179.166,5.357,148.679
C00615=1230.082,28.391,-42.790,-179.164,5.356,148.679
C00616=1230.077,28.640,-42.805,-179.161,5.357,148.678
C00617=1230.072,28.889,-42.822,-179.158,5.358,148.677
C00618=1230.067,29.139,-42.838,-179.156,5.358,148.677
C00619=1230.062,29.407,-42.854,-179.153,5.359,148.676
C00620=1230.057,29.676,-42.871,-179.150,5.359,148.675
C00621=1230.051,29.945,-42.887,-179.147,5.359,148.674
C00622=1230.045,30.214,-42.904,-179.145,5.360,148.674
C00623=1230.041,30.463,-42.921,-179.142,5.361,148.673
C00624=1230.036,30.712,-42.936,-179.140,5.360,148.672
C00625=1230.031,30.962,-42.952,-179.137,5.361,148.672
C00626=1230.026,31.212,-42.968,-179.135,5.361,148.671
C00627=1230.021,31.461,-42.983,-179.133,5.362,148.671
C00628=1230.016,31.711,-43.000,-179.130,5.363,148.670
C00629=1230.011,31.960,-43.015,-179.127,5.363,148.669
C00630=1230.006,32.209,-43.031,-179.125,5.363,148.669
C00631=1230.001,32.459,-43.046,-179.123,5.364,148.668
C00632=1229.996,32.708,-43.063,-179.120,5.364,148.667
C00633=1229.991,32.957,-43.078,-179.117,5.365,148.667
C00634=1229.986,33.207,-43.094,-179.115,5.365,148.666
C00635=1229.981,33.456,-43.111,-179.112,5.366,148.665
C00636=1229.977,33.706,-43.126,-179.109,5.366,148.665
C00637=1229.972,33.955,-43.142,-179.107,5.366,148.664
C00638=1229.966,34.205,-43.157,-179.105,5.367,148.663
C00639=1229.962,34.454,-43.174,-179.102,5.367,148.662
C00640=1229.956,34.704,-43.189,-179.099,5.368,148.662
C00641=1229.951,34.954,-43.205,-179.097,5.368,148.661
C00642=1229.946,35.203,-43.222,-179.094,5.369,148.660
C00643=1229.941,35.452,-43.237,-179.092,5.369,148.660
C00644=1229.937,35.701,-43.253,-179.090,5.370,148.659
C00645=1229.932,35.951,-43.269,-179.087,5.370,148.659
C00646=1229.927,36.201,-43.285,-179.085,5.371,148.658
C00647=1229.922,36.449,-43.301,-179.082,5.371,148.657
C00648=1229.917,36.700,-43.317,-179.079,5.372,148.657
C00649=1229.912,36.949,-43.333,-179.077,5.372,148.656
C00650=1229.907,37.198,-43.349,-179.075,5.372,148.655
C00651=1229.902,37.448,-43.365,-179.072,5.373,148.655
C00652=1229.897,37.697,-43.381,-179.069,5.373,148.654
C00653=1229.892,37.947,-43.397,-179.067,5.374,148.653
C00654=1229.887,38.195,-43.414,-179.064,5.374,148.653
C00655=1229.882,38.446,-43.429,-179.061,5.375,148.652
C00656=1229.877,38.694,-43.446,-179.059,5.376,148.651
C00657=1229.872,38.944,-43.462,-179.057,5.375,148.651
C00658=1229.867,39.194,-43.477,-179.054,5.376,148.650
C00659=1229.862,39.443,-43.494,-179.052,5.377,148.649
C00660=1229.857,39.693,-43.510,-179.049,5.377,148.649
C00661=1229.852,39.942,-43.526,-179.047,5.378,148.648
C00662=1229.847,40.192,-43.542,-179.044,5.378,148.647
C00663=1229.842,40.440,-43.558,-179.041,5.379,148.647
C00664=1229.838,40.690,-43.575,-179.039,5.380,148.646
C00665=1229.832,40.939,-43.590,-179.037,5.379,148.645
C00666=1229.828,41.189,-43.607,-179.034,5.380,148.645
C00667=1229.822,41.438,-43.623,-179.031,5.380,148.644
C00668=1229.818,41.688,-43.639,-179.029,5.381,148.643
C00669=1229.813,41.937,-43.655,-179.026,5.382,148.643
C00670=1229.808,42.187,-43.672,-179.023,5.382,148.642
C00671=1229.803,42.436,-43.687,-179.021,5.383,148.642
C00672=1229.798,42.685,-43.704,-179.019,5.384,148.641
C00673=1229.794,42.935,-43.721,-179.016,5.384,148.640
C00674=1229.788,43.185,-43.737,-179.014,5.384,148.640
C00675=1229.783,43.434,-43.753,-179.011,5.385,148.639
C00676=1229.778,43.684,-43.769,-179.009,5.385,148.638
C00677=1229.773,43.933,-43.786,-179.006,5.386,148.638
C00678=1229.768,44.182,-43.802,-179.003,5.386,148.637
C00679=1229.763,44.432,-43.818,-179.001,5.387,148.636
C00680=1229.758,44.681,-43.834,-178.998,5.387,148.636
C00681=1229.754,44.930,-43.851,-178.995,5.388,148.635
C00682=1229.748,45.180,-43.866,-178.993,5.389,148.634
C00683=1229.743,45.429,-43.884,-178.991,5.389,148.634
C00684=1229.739,45.679,-43.900,-178.989,5.389,148.633
C00685=1229.733,45.928,-43.916,-178.986,5.390,148.632
C00686=1229.729,46.178,-43.933,-178.983,5.390,148.632
C00687=1229.724,46.427,-43.949,-178.981,5.391,148.631
C00688=1229.719,46.676,-43.966,-178.978,5.391,148.630
C00689=1229.714,46.925,-43.981,-178.975,5.392,148.630
C00690=1229.709,47.175,-43.998,-178.973,5.393,148.629
C00691=1229.704,47.425,-44.015,-178.970,5.393,148.628
C00692=1229.699,47.673,-44.031,-178.968,5.394,148.628
C00693=1229.694,47.924,-44.047,-178.966,5.394,148.627
C00694=1229.689,48.172,-44.064,-178.963,5.394,148.627
C00695=1229.684,48.422,-44.081,-178.961,5.395,148.626
C00696=1229.680,48.672,-44.098,-178.958,5.396,148.625
C00697=1229.675,48.920,-44.114,-178.955,5.396,148.625
C00698=1229.670,49.171,-44.130,-178.953,5.397,148.624
C00699=1229.665,49.420,-44.147,-178.950,5.397,148.623
C00700=1229.659,49.669,-44.163,-178.947,5.398,148.623
C00701=1229.655,49.919,-44.180,-178.945,5.398,148.622
C00702=1229.650,50.167,-44.196,-178.943,5.399,148.621
C00703=1229.645,50.417,-44.212,-178.940,5.400,148.621
C00704=1229.640,50.667,-44.230,-178.938,5.400,148.620
C00705=1229.635,50.916,-44.246,-178.935,5.400,148.619
C00706=1229.630,51.166,-44.263,-178.933,5.401,148.619
C00707=1229.626,51.415,-44.279,-178.930,5.401,148.618
C00708=1229.620,51.664,-44.296,-178.927,5.402,148.617
C00709=1229.616,51.914,-44.313,-178.925,5.402,148.617
C00710=1229.611,52.163,-44.330,-178.923,5.403,148.616
C00711=1229.606,52.412,-44.346,-178.920,5.404,148.616
C00712=1229.601,52.662,-44.363,-178.917,5.405,148.615
C00713=1229.596,52.912,-44.379,-178.915,5.405,148.614
C00714=1229.591,53.161,-44.395,-178.912,5.406,148.614
C00715=1229.586,53.410,-44.413,-178.909,5.406,148.613
C00716=1229.581,53.660,-44.429,-178.907,5.407,148.612
C00717=1229.576,53.909,-44.446,-178.904,5.407,148.612
C00718=1229.571,54.158,-44.463,-178.902,5.407,148.611
C00719=1229.566,54.408,-44.480,-178.900,5.408,148.611
C00720=1229.562,54.657,-44.496,-178.897,5.409,148.610
C00721=1229.556,54.906,-44.513,-178.895,5.409,148.609
C00722=1229.552,55.156,-44.530,-178.892,5.410,148.609
C00723=1229.546,55.424,-44.548,-178.889,5.410,148.608
C00724=1229.541,55.693,-44.566,-178.887,5.411,148.607
C00725=1229.536,55.961,-44.584,-178.884,5.412,148.607
C00726=1229.530,56.229,-44.603,-178.881,5.413,148.606
C00727=1229.526,56.479,-44.619,-178.879,5.413,148.605
C00728=1229.520,56.728,-44.636,-178.876,5.413,148.605
C00729=1229.516,56.977,-44.653,-178.874,5.414,148.604
C00730=1229.511,57.227,-44.670,-178.871,5.414,148.603
C00731=1229.506,57.477,-44.687,-178.868,5.415,148.602
C00732=1229.501,57.726,-44.703,-178.866,5.416,148.602
C00733=1229.496,57.975,-44.720,-178.864,5.416,148.601
C00734=1229.491,58.225,-44.737,-178.861,5.417,148.601
C00735=1229.486,58.475,-44.754,-178.858,5.418,148.600
C00736=1229.481,58.723,-44.771,-178.856,5.418,148.599
C00737=1229.477,58.972,-44.788,-178.853,5.419,148.599
C00738=1229.471,59.222,-44.805,-178.850,5.419,148.598
C00739=1229.467,59.472,-44.822,-178.848,5.420,148.597
C00740=1229.462,59.721,-44.839,-178.846,5.421,148.597
C00741=1229.457,59.970,-44.855,-178.843,5.421,148.596
C00742=1229.452,60.219,-44.873,-178.840,5.422,148.596
C00743=1229.447,60.469,-44.890,-178.838,5.423,148.595
C00744=1229.442,60.719,-44.907,-178.835,5.423,148.594
C00745=1229.437,60.967,-44.924,-178.832,5.424,148.594
C00746=1229.432,61.217,-44.941,-178.830,5.424,148.593
C00747=1229.428,61.466,-44.958,-178.828,5.425,148.593
C00748=1229.422,61.716,-44.976,-178.825,5.426,148.592
C00749=1229.418,61.965,-44.992,-178.822,5.426,148.591
C00750=1229.412,62.214,-45.009,-178.820,5.427,148.591
C00751=1229.408,62.464,-45.026,-178.817,5.428,148.590
C00752=1229.403,62.713,-45.044,-178.815,5.427,148.589
C00753=1229.398,62.963,-45.060,-178.813,5.428,148.589
C00754=1229.393,63.212,-45.078,-178.810,5.429,148.588
C00755=1229.388,63.462,-45.096,-178.808,5.429,148.587
C00756=1229.383,63.710,-45.112,-178.805,5.430,148.587
C00757=1229.378,63.960,-45.129,-178.802,5.431,148.586
C00758=1229.373,64.210,-45.146,-178.800,5.431,148.585
C00759=1229.368,64.459,-45.164,-178.797,5.432,148.585
C00760=1229.364,64.708,-45.181,-178.795,5.433,148.584
C00761=1229.359,64.958,-45.198,-178.792,5.433,148.584
C00762=1229.354,65.207,-45.216,-178.790,5.434,148.583
C00763=1229.349,65.456,-45.232,-178.787,5.434,148.582
C00764=1229.344,65.705,-45.250,-178.785,5.435,148.582
C00765=1229.339,65.955,-45.267,-178.782,5.436,148.581
C00766=1229.334,66.204,-45.284,-178.780,5.437,148.581
C00767=1229.329,66.454,-45.302,-178.777,5.437,148.580
C00768=1229.325,66.703,-45.319,-178.774,5.438,148.579
C00769=1229.319,66.953,-45.336,-178.772,5.438,148.579
C00770=1229.315,67.202,-45.354,-178.769,5.439,148.578
C00771=1229.310,67.452,-45.371,-178.767,5.440,148.577
C00772=1229.305,67.700,-45.388,-178.764,5.440,148.577
C00773=1229.300,67.950,-45.405,-178.762,5.441,148.576
C00774=1229.295,68.199,-45.423,-178.759,5.442,148.576
C00775=1229.290,68.448,-45.440,-178.757,5.442,148.575
C00776=1229.286,68.697,-45.458,-178.754,5.443,148.574
C00777=1229.281,68.947,-45.475,-178.752,5.444,148.574
C00778=1229.275,69.197,-45.492,-178.749,5.444,148.573
C00779=1229.270,69.446,-45.510,-178.747,5.445,148.572
C00780=1229.266,69.696,-45.527,-178.744,5.445,148.572
C00781=1229.261,69.945,-45.545,-178.741,5.446,148.571
C00782=1229.256,70.194,-45.563,-178.739,5.447,148.570
C00783=1229.252,70.443,-45.579,-178.737,5.448,148.570
C00784=1229.247,70.693,-45.597,-178.734,5.448,148.569
C00785=1229.241,70.942,-45.615,-178.731,5.449,148.569
C00786=1229.236,71.191,-45.632,-178.729,5.449,148.568
C00787=1229.231,71.440,-45.649,-178.726,5.450,148.567
C00788=1229.227,71.690,-45.667,-178.724,5.451,148.567
C00789=1229.221,71.939,-45.684,-178.721,5.451,148.566
C00790=1229.216,72.189,-45.702,-178.719,5.452,148.566
C00791=1229.212,72.437,-45.719,-178.716,5.453,148.565
C00792=1229.207,72.687,-45.737,-178.713,5.453,148.564
C00793=1229.202,72.936,-45.755,-178.711,5.454,148.564
C00794=1229.197,73.186,-45.772,-178.709,5.455,148.563
C00795=1229.193,73.435,-45.789,-178.706,5.455,148.563
C00796=1229.188,73.684,-45.807,-178.703,5.457,148.562
C00797=1229.183,73.934,-45.825,-178.700,5.457,148.561
C00798=1229.178,74.183,-45.843,-178.698,5.458,148.561
C00799=1229.173,74.432,-45.861,-178.695,5.459,148.560
C00800=1229.168,74.682,-45.877,-178.693,5.460,148.560
C00801=1229.163,74.931,-45.895,-178.690,5.460,148.559
C00802=1229.158,75.180,-45.913,-178.687,5.461,148.558
C00803=1229.153,75.430,-45.930,-178.685,5.462,148.558
C00804=1229.148,75.679,-45.948,-178.683,5.462,148.557
C00805=1229.143,75.928,-45.966,-178.680,5.463,148.556
C00806=1229.138,76.178,-45.984,-178.677,5.463,148.556
C00807=1229.134,76.427,-46.001,-178.675,5.464,148.555
C00808=1229.129,76.676,-46.019,-178.673,5.465,148.555
C00809=1229.124,76.925,-46.037,-178.670,5.466,148.554
C00810=1229.120,77.176,-46.055,-178.667,5.466,148.553
C00811=1229.115,77.425,-46.073,-178.665,5.467,148.553
C00812=1229.110,77.674,-46.091,-178.662,5.467,148.552
C00813=1229.105,77.923,-46.109,-178.660,5.468,148.552
C00814=1229.100,78.173,-46.127,-178.657,5.469,148.551
C00815=1229.095,78.422,-46.143,-178.655,5.469,148.550
C00816=1229.091,78.671,-46.161,-178.652,5.470,148.550
C00817=1229.086,78.920,-46.179,-178.650,5.471,148.549
C00818=1229.081,79.170,-46.197,-178.647,5.472,148.549
C00819=1229.076,79.419,-46.215,-178.645,5.472,148.548
C00820=1229.071,79.669,-46.232,-178.642,5.474,148.547
C00821=1229.066,79.918,-46.250,-178.639,5.474,148.547
C00822=1229.061,80.167,-46.268,-178.637,5.475,148.546
C00823=1229.056,80.416,-46.286,-178.634,5.476,148.546
C00824=1229.052,80.666,-46.305,-178.632,5.476,148.545
C00825=1229.047,80.915,-46.323,-178.629,5.477,148.544
C00826=1229.042,81.164,-46.341,-178.627,5.478,148.544
C00827=1229.036,81.433,-46.359,-178.624,5.478,148.543
C00828=1229.031,81.701,-46.379,-178.622,5.479,148.542
C00829=1229.026,81.970,-46.398,-178.618,5.480,148.542
C00830=1229.021,82.238,-46.418,-178.616,5.481,148.541
C00831=1229.016,82.487,-46.436,-178.613,5.482,148.541
C00832=1229.011,82.736,-46.454,-178.611,5.482,148.540
C00833=1229.006,82.985,-46.472,-178.608,5.483,148.539
C00834=1229.001,83.235,-46.490,-178.606,5.484,148.539
C00835=1228.997,83.484,-46.508,-178.603,5.484,148.538
C00836=1228.992,83.733,-46.525,-178.601,5.485,148.537
C00837=1228.987,83.983,-46.544,-178.598,5.486,148.537
C00838=1228.982,84.232,-46.562,-178.596,5.487,148.536
C00839=1228.977,84.481,-46.580,-178.593,5.487,148.536
C00840=1228.972,84.731,-46.598,-178.590,5.489,148.535
C00841=1228.967,84.980,-46.616,-178.587,5.489,148.534
C00842=1228.962,85.229,-46.634,-178.585,5.490,148.534
C00843=1228.958,85.479,-46.653,-178.583,5.491,148.533
C00844=1228.953,85.728,-46.671,-178.580,5.491,148.533
C00845=1228.948,85.977,-46.689,-178.577,5.492,148.532
C00846=1228.943,86.226,-46.707,-178.575,5.493,148.532
C00847=1228.938,86.476,-46.725,-178.573,5.493,148.531
C00848=1228.934,86.725,-46.743,-178.570,5.494,148.530
C00849=1228.928,86.975,-46.762,-178.567,5.495,148.530
C00850=1228.923,87.224,-46.779,-178.565,5.496,148.529
C00851=1228.919,87.473,-46.798,-178.562,5.497,148.529
C00852=1228.914,87.722,-46.816,-178.559,5.498,148.528
C00853=1228.909,87.972,-46.835,-178.557,5.498,148.527
C00854=1228.904,88.221,-46.852,-178.555,5.499,148.527
C00855=1228.900,88.470,-46.870,-178.552,5.500,148.526
C00856=1228.895,88.719,-46.888,-178.549,5.500,148.526
C00857=1228.889,88.969,-46.907,-178.547,5.501,148.525
C00858=1228.885,89.218,-46.926,-178.545,5.502,148.524
C00859=1228.880,89.467,-46.944,-178.542,5.503,148.524
C00860=1228.875,89.716,-46.962,-178.539,5.503,148.523
C00861=1228.870,89.966,-46.980,-178.536,5.505,148.523
C00862=1228.865,90.216,-46.999,-178.534,5.506,148.522
C00863=1228.861,90.464,-47.018,-178.531,5.506,148.521
C00864=1228.856,90.713,-47.036,-178.529,5.507,148.521
C00865=1228.851,90.963,-47.054,-178.527,5.508,148.520
C00866=1228.846,91.213,-47.072,-178.524,5.508,148.520
C00867=1228.841,91.461,-47.091,-178.521,5.509,148.519
C00868=1228.836,91.711,-47.109,-178.519,5.510,148.518
C00869=1228.832,91.960,-47.128,-178.517,5.510,148.518
C00870=1228.827,92.210,-47.146,-178.514,5.512,148.517
C00871=1228.822,92.458,-47.165,-178.511,5.513,148.517
C00872=1228.817,92.708,-47.183,-178.508,5.513,148.516
C00873=1228.812,92.958,-47.201,-178.506,5.514,148.516
C00874=1228.808,93.206,-47.220,-178.504,5.515,148.515
C00875=1228.802,93.456,-47.238,-178.501,5.515,148.514
C00876=1228.798,93.705,-47.257,-178.499,5.516,148.514
C00877=1228.793,93.954,-47.275,-178.496,5.517,148.513
C00878=1228.788,94.203,-47.294,-178.493,5.518,148.513
C00879=1228.783,94.453,-47.312,-178.490,5.519,148.512
C00880=1228.779,94.702,-47.331,-178.488,5.520,148.512
C00881=1228.774,94.951,-47.349,-178.486,5.520,148.511
C00882=1228.768,95.201,-47.368,-178.483,5.521,148.510
C00883=1228.764,95.450,-47.387,-178.481,5.522,148.510
C00884=1228.759,95.699,-47.405,-178.478,5.523,148.509
C00885=1228.754,95.948,-47.424,-178.475,5.524,148.509
C00886=1228.750,96.198,-47.442,-178.473,5.525,148.508
C00887=1228.745,96.446,-47.461,-178.470,5.526,148.507
C00888=1228.739,96.696,-47.480,-178.468,5.526,148.507
C00889=1228.735,96.946,-47.498,-178.465,5.527,148.506
C00890=1228.730,97.195,-47.517,-178.463,5.528,148.506
C00891=1228.725,97.444,-47.536,-178.460,5.528,148.505
C00892=1228.721,97.693,-47.554,-178.457,5.530,148.504
C00893=1228.715,97.942,-47.573,-178.455,5.531,148.504
C00894=1228.711,98.192,-47.592,-178.452,5.531,148.503
C00895=1228.706,98.441,-47.610,-178.450,5.532,148.503
C00896=1228.701,98.690,-47.629,-178.448,5.533,148.502
C00897=1228.696,98.940,-47.648,-178.445,5.534,148.502
C00898=1228.691,99.189,-47.667,-178.442,5.534,148.501
C00899=1228.687,99.438,-47.685,-178.440,5.536,148.501
C00900=1228.681,99.687,-47.704,-178.437,5.537,148.500
C00901=1228.677,99.936,-47.723,-178.435,5.537,148.499
C00902=1228.673,100.186,-47.742,-178.432,5.538,148.499
C00903=1228.667,100.435,-47.761,-178.430,5.539,148.498
C00904=1228.663,100.684,-47.779,-178.427,5.539,148.498
C00905=1228.658,100.933,-47.798,-178.424,5.541,148.497
C00906=1228.653,101.182,-47.816,-178.422,5.542,148.497
C00907=1228.648,101.432,-47.836,-178.419,5.542,148.496
C00908=1228.643,101.681,-47.855,-178.417,5.543,148.495
C00909=1228.638,101.931,-47.874,-178.415,5.544,148.495
C00910=1228.634,102.179,-47.892,-178.412,5.545,148.494
C00911=1228.629,102.429,-47.912,-178.409,5.546,148.494
C00912=1228.624,102.678,-47.930,-178.407,5.547,148.493
C00913=1228.619,102.928,-47.950,-178.404,5.548,148.493
C00914=1228.615,103.176,-47.968,-178.401,5.548,148.492
C00915=1228.609,103.426,-47.987,-178.399,5.549,148.491
C00916=1228.605,103.675,-48.006,-178.396,5.551,148.491
C00917=1228.600,103.924,-48.025,-178.393,5.551,148.490
C00918=1228.595,104.174,-48.044,-178.391,5.552,148.490
C00919=1228.590,104.423,-48.063,-178.389,5.553,148.489
C00920=1228.586,104.672,-48.082,-178.386,5.553,148.488
C00921=1228.581,104.921,-48.101,-178.384,5.554,148.488
C00922=1228.576,105.171,-48.120,-178.381,5.556,148.487
C00923=1228.571,105.419,-48.139,-178.378,5.556,148.487
C00924=1228.566,105.669,-48.159,-178.376,5.557,148.486
C00925=1228.562,105.918,-48.177,-178.373,5.558,148.486
C00926=1228.557,106.168,-48.196,-178.371,5.559,148.485
C00927=1228.552,106.416,-48.215,-178.368,5.560,148.485
C00928=1228.547,106.666,-48.235,-178.366,5.561,148.484
C00929=1228.542,106.915,-48.254,-178.363,5.562,148.483
C00930=1228.538,107.164,-48.273,-178.361,5.563,148.483
C00931=1228.532,107.433,-48.293,-178.358,5.564,148.482
C00932=1228.527,107.701,-48.314,-178.355,5.565,148.482
C00933=1228.522,107.969,-48.335,-178.352,5.565,148.481
C00934=1228.516,108.238,-48.355,-178.349,5.567,148.480
C00935=1228.512,108.487,-48.374,-178.347,5.568,148.480
C00936=1228.507,108.737,-48.393,-178.344,5.568,148.479
C00937=1228.502,108.986,-48.413,-178.342,5.569,148.479
C00938=1228.498,109.235,-48.432,-178.339,5.571,148.478
C00939=1228.493,109.484,-48.451,-178.337,5.571,148.478
C00940=1228.488,109.733,-48.471,-178.334,5.572,148.477
C00941=1228.484,109.982,-48.490,-178.332,5.573,148.477
C00942=1228.478,110.231,-48.509,-178.329,5.574,148.476
C00943=1228.474,110.481,-48.529,-178.327,5.575,148.476
C00944=1228.469,110.730,-48.547,-178.324,5.576,148.475
C00945=1228.464,110.980,-48.566,-178.321,5.577,148.474
C00946=1228.459,111.229,-48.586,-178.319,5.578,148.474
C00947=1228.454,111.478,-48.605,-178.316,5.579,148.473
C00948=1228.450,111.727,-48.624,-178.314,5.580,148.473
C00949=1228.444,111.976,-48.644,-178.311,5.581,148.472
C00950=1228.440,112.226,-48.663,-178.309,5.581,148.472
C00951=1228.435,112.475,-48.683,-178.307,5.582,148.471
C00952=1228.430,112.724,-48.702,-178.303,5.584,148.471
C00953=1228.426,112.973,-48.721,-178.301,5.584,148.470
C00954=1228.420,113.222,-48.741,-178.299,5.585,148.469
C00955=1228.416,113.471,-48.761,-178.296,5.586,148.469
C00956=1228.412,113.720,-48.780,-178.293,5.588,148.468
C00957=1228.406,113.969,-48.799,-178.291,5.588,148.468
C00958=1228.402,114.219,-48.819,-178.288,5.589,148.467
C00959=1228.396,114.468,-48.838,-178.286,5.590,148.467
C00960=1228.392,114.717,-48.858,-178.283,5.591,148.466
C00961=1228.388,114.967,-48.877,-178.281,5.592,148.466
C00962=1228.382,115.215,-48.896,-178.278,5.593,148.465
C00963=1228.378,115.465,-48.916,-178.275,5.594,148.464
C00964=1228.373,115.715,-48.936,-178.273,5.595,148.464
C00965=1228.367,115.963,-48.955,-178.270,5.596,148.463
C00966=1228.363,116.212,-48.975,-178.268,5.597,148.463
C00967=1228.359,116.462,-48.994,-178.265,5.598,148.462
C00968=1228.354,116.711,-49.014,-178.262,5.599,148.462
C00969=1228.349,116.960,-49.033,-178.260,5.600,148.461
C00970=1228.344,117.210,-49.053,-178.258,5.601,148.461
C00971=1228.339,117.459,-49.072,-178.255,5.601,148.460
C00972=1228.334,117.707,-49.093,-178.252,5.603,148.460
C00973=1228.330,117.957,-49.112,-178.250,5.604,148.459
C00974=1228.324,118.206,-49.132,-178.248,5.605,148.459
C00975=1228.320,118.455,-49.151,-178.245,5.605,148.458
C00976=1228.316,118.704,-49.171,-178.242,5.607,148.458
C00977=1228.311,118.954,-49.191,-178.240,5.608,148.457
C00978=1228.306,119.203,-49.210,-178.237,5.608,148.456
C00979=1228.301,119.452,-49.230,-178.235,5.609,148.456
C00980=1228.297,119.701,-49.250,-178.232,5.611,148.455
C00981=1228.291,119.950,-49.269,-178.230,5.612,148.455
C00982=1228.287,120.200,-49.289,-178.227,5.612,148.454
C00983=1228.282,120.448,-49.309,-178.224,5.613,148.454
C00984=1228.277,120.698,-49.329,-178.222,5.615,148.453
C00985=1228.272,120.947,-49.348,-178.219,5.615,148.453
C00986=1228.267,121.196,-49.368,-178.217,5.616,148.452
C00987=1228.263,121.445,-49.388,-178.214,5.618,148.452
C00988=1228.258,121.695,-49.408,-178.212,5.619,148.451
C00989=1228.253,121.943,-49.428,-178.209,5.619,148.450
C00990=1228.248,122.193,-49.448,-178.206,5.620,148.450
C00991=1228.244,122.442,-49.467,-178.204,5.622,148.449
C00992=1228.239,122.691,-49.488,-178.201,5.622,148.449
C00993=1228.234,122.940,-49.507,-178.199,5.623,148.448
C00994=1228.229,123.190,-49.527,-178.196,5.625,148.448
C00995=1228.225,123.439,-49.547,-178.194,5.626,148.447
C00996=1228.220,123.688,-49.567,-178.191,5.626,148.447
C00997=1228.215,123.936,-49.587,-178.189,5.627,148.446
C00998=1228.210,124.186,-49.606,-178.186,5.629,148.446
C00999=1228.206,124.435,-49.627,-178.183,5.630,148.445
C01000=1228.201,124.685,-49.646,-178.181,5.631,148.445
C01001=1228.196,124.934,-49.667,-178.178,5.632,148.444
C01002=1228.191,125.182,-49.686,-178.176,5.633,148.444
C01003=1228.187,125.431,-49.706,-178.173,5.634,148.443
C01004=1228.182,125.681,-49.726,-178.171,5.635,148.443
C01005=1228.178,125.930,-49.746,-178.168,5.636,148.442
C01006=1228.173,126.179,-49.766,-178.165,5.637,148.441
C01007=1228.168,126.429,-49.787,-178.163,5.638,148.441
C01008=1228.162,126.678,-49.806,-178.160,5.639,148.440
C01009=1228.158,126.927,-49.827,-178.158,5.640,148.440
C01010=1228.153,127.176,-49.846,-178.155,5.641,148.439
C01011=1228.149,127.425,-49.867,-178.153,5.642,148.439
C01012=1228.144,127.675,-49.886,-178.150,5.643,148.438
C01013=1228.139,127.924,-49.907,-178.148,5.644,148.438
C01014=1228.134,128.172,-49.927,-178.145,5.646,148.437
C01015=1228.129,128.422,-49.947,-178.143,5.647,148.437
C01016=1228.124,128.671,-49.967,-178.140,5.647,148.436
C01017=1228.120,128.920,-49.987,-178.137,5.649,148.436
C01018=1228.115,129.169,-50.007,-178.135,5.650,148.435
C01019=1228.111,129.418,-50.028,-178.132,5.650,148.435
C01020=1228.106,129.668,-50.047,-178.130,5.652,148.434
C01021=1228.101,129.917,-50.068,-178.127,5.653,148.434
C01022=1228.096,130.165,-50.088,-178.125,5.654,148.433
C01023=1228.091,130.415,-50.108,-178.122,5.655,148.432
C01024=1228.087,130.664,-50.128,-178.120,5.656,148.432
C01025=1228.082,130.913,-50.149,-178.117,5.657,148.431
C01026=1228.077,131.163,-50.169,-178.114,5.659,148.431
C01027=1228.072,131.411,-50.189,-178.112,5.659,148.430
C01028=1228.068,131.660,-50.210,-178.110,5.660,148.430
C01029=1228.064,131.909,-50.230,-178.106,5.662,148.429
C01030=1228.058,132.159,-50.250,-178.104,5.663,148.429
C01031=1228.054,132.408,-50.271,-178.102,5.663,148.428
C01032=1228.049,132.656,-50.291,-178.099,5.665,148.428
C01033=1228.044,132.905,-50.311,-178.096,5.666,148.427
C01034=1228.039,133.155,-50.331,-178.094,5.667,148.427
C01035=1228.035,133.424,-50.354,-178.091,5.668,148.426
C01036=1228.029,133.693,-50.375,-178.089,5.669,148.426
C01037=1228.024,133.961,-50.398,-178.085,5.670,148.425
C01038=1228.019,134.229,-50.419,-178.083,5.671,148.425
C01039=1228.014,134.479,-50.440,-178.080,5.673,148.424
C01040=1228.009,134.728,-50.460,-178.078,5.674,148.424
C01041=1228.005,134.977,-50.480,-178.075,5.675,148.423
C01042=1227.999,135.226,-50.501,-178.073,5.676,148.423
C01043=1227.995,135.475,-50.522,-178.070,5.677,148.422
C01044=1227.991,135.724,-50.542,-178.067,5.679,148.422
C01045=1227.985,135.974,-50.563,-178.065,5.679,148.421
C01046=1227.981,136.223,-50.583,-178.063,5.680,148.421
C01047=1227.976,136.472,-50.604,-178.060,5.682,148.420
C01048=1227.971,136.721,-50.624,-178.057,5.683,148.420
C01049=1227.967,136.970,-50.644,-178.055,5.683,148.419
C01050=1227.961,137.220,-50.665,-178.052,5.685,148.419
C01051=1227.957,137.468,-50.686,-178.050,5.686,148.418
C01052=1227.953,137.717,-50.706,-178.047,5.688,148.418
C01053=1227.947,137.967,-50.727,-178.044,5.688,148.417
C01054=1227.943,138.216,-50.748,-178.042,5.689,148.417
C01055=1227.938,138.465,-50.768,-178.039,5.691,148.416
C01056=1227.933,138.714,-50.789,-178.037,5.692,148.416
C01057=1227.929,138.963,-50.809,-178.034,5.692,148.415
C01058=1227.924,139.212,-50.830,-178.032,5.694,148.415
C01059=1227.919,139.461,-50.851,-178.029,5.695,148.414
C01060=1227.914,139.710,-50.872,-178.026,5.697,148.414
C01061=1227.910,139.959,-50.892,-178.024,5.697,148.413
C01062=1227.905,140.208,-50.913,-178.022,5.698,148.412
C01063=1227.900,140.457,-50.933,-178.019,5.700,148.412
C01064=1227.895,140.707,-50.954,-178.016,5.701,148.411
C01065=1227.891,140.956,-50.975,-178.014,5.702,148.411
C01066=1227.886,141.206,-50.996,-178.011,5.703,148.410
C01067=1227.881,141.455,-51.016,-178.009,5.704,148.410
C01068=1227.877,141.703,-51.038,-178.006,5.706,148.409
C01069=1227.872,141.952,-51.058,-178.004,5.706,148.409
C01070=1227.867,142.201,-51.079,-178.001,5.708,148.408
C01071=1227.863,142.450,-51.100,-177.999,5.709,148.408
C01072=1227.857,142.700,-51.121,-177.996,5.710,148.407
C01073=1227.853,142.949,-51.141,-177.993,5.711,148.407
C01074=1227.848,143.198,-51.162,-177.991,5.712,148.406
C01075=1227.844,143.446,-51.183,-177.988,5.714,148.406
C01076=1227.839,143.696,-51.204,-177.986,5.715,148.406
C01077=1227.835,143.945,-51.225,-177.983,5.716,148.405
C01078=1227.829,144.194,-51.246,-177.981,5.717,148.405
C01079=1227.825,144.443,-51.266,-177.978,5.718,148.404
C01080=1227.820,144.692,-51.288,-177.975,5.720,148.404
C01081=1227.815,144.941,-51.309,-177.973,5.720,148.403
C01082=1227.811,145.190,-51.329,-177.971,5.721,148.403
C01083=1227.805,145.439,-51.350,-177.967,5.723,148.402
C01084=1227.802,145.688,-51.372,-177.965,5.724,148.402
C01085=1227.797,145.938,-51.393,-177.963,5.726,148.401
C01086=1227.791,146.187,-51.413,-177.960,5.726,148.401
C01087=1227.787,146.436,-51.434,-177.957,5.728,148.400
C01088=1227.782,146.684,-51.456,-177.955,5.729,148.400
C01089=1227.778,146.933,-51.476,-177.953,5.730,148.399
C01090=1227.773,147.183,-51.497,-177.950,5.731,148.399
C01091=1227.768,147.432,-51.519,-177.947,5.732,148.398
C01092=1227.764,147.681,-51.539,-177.944,5.734,148.398
C01093=1227.759,147.930,-51.560,-177.942,5.735,148.397
C01094=1227.754,148.179,-51.582,-177.940,5.737,148.397
C01095=1227.749,148.428,-51.602,-177.937,5.737,148.396
C01096=1227.745,148.678,-51.624,-177.934,5.739,148.396
C01097=1227.740,148.926,-51.645,-177.932,5.740,148.395
C01098=1227.735,149.175,-51.666,-177.930,5.741,148.395
C01099=1227.731,149.424,-51.687,-177.926,5.742,148.394
C01100=1227.725,149.673,-51.708,-177.924,5.743,148.394
C01101=1227.721,149.923,-51.730,-177.922,5.745,148.393
C01102=1227.717,150.172,-51.751,-177.919,5.746,148.393
C01103=1227.712,150.421,-51.772,-177.916,5.747,148.392
C01104=1227.707,150.669,-51.793,-177.914,5.748,148.392
C01105=1227.702,150.918,-51.814,-177.911,5.750,148.391
C01106=1227.698,151.168,-51.836,-177.909,5.751,148.391
C01107=1227.693,151.417,-51.857,-177.906,5.752,148.390
C01108=1227.688,151.666,-51.879,-177.904,5.753,148.390
C01109=1227.683,151.915,-51.899,-177.901,5.754,148.389
C01110=1227.679,152.164,-51.921,-177.899,5.756,148.389
C01111=1227.674,152.413,-51.942,-177.896,5.757,148.389
C01112=1227.669,152.662,-51.964,-177.893,5.758,148.388
C01113=1227.664,152.911,-51.985,-177.891,5.759,148.388
C01114=1227.660,153.160,-52.006,-177.888,5.761,148.387
C01115=1227.655,153.409,-52.027,-177.886,5.762,148.387
C01116=1227.650,153.658,-52.049,-177.883,5.764,148.386
C01117=1227.645,153.907,-52.070,-177.881,5.764,148.386
C01118=1227.641,154.157,-52.092,-177.878,5.766,148.385
C01119=1227.636,154.405,-52.113,-177.875,5.767,148.385
C01120=1227.632,154.654,-52.134,-177.873,5.769,148.384
C01121=1227.627,154.904,-52.156,-177.871,5.770,148.384
C01122=1227.623,155.152,-52.177,-177.868,5.770,148.383
C01123=1227.617,155.401,-52.198,-177.865,5.772,148.383
C01124=1227.613,155.651,-52.220,-177.863,5.773,148.382
C01125=1227.608,155.900,-52.241,-177.860,5.774,148.382
C01126=1227.603,156.149,-52.263,-177.858,5.775,148.382
C01127=1227.599,156.397,-52.284,-177.855,5.777,148.381
C01128=1227.594,156.647,-52.306,-177.853,5.778,148.381
C01129=1227.590,156.896,-52.327,-177.850,5.780,148.380
C01130=1227.585,157.144,-52.349,-177.848,5.780,148.380
C01131=1227.580,157.394,-52.371,-177.845,5.782,148.379
C01132=1227.575,157.643,-52.392,-177.842,5.783,148.379
C01133=1227.570,157.892,-52.414,-177.840,5.785,148.378
C01134=1227.566,158.141,-52.436,-177.838,5.786,148.378
C01135=1227.561,158.389,-52.457,-177.834,5.787,148.377
C01136=1227.557,158.639,-52.479,-177.832,5.788,148.377
C01137=1227.552,158.888,-52.500,-177.830,5.790,148.376
C01138=1227.547,159.137,-52.522,-177.827,5.791,148.376
C01139=1227.542,159.406,-52.545,-177.824,5.793,148.376
C01140=1227.537,159.675,-52.569,-177.821,5.794,148.375
C01141=1227.531,159.944,-52.592,-177.819,5.795,148.375
C01142=1227.527,160.214,-52.615,-177.816,5.796,148.374
C01143=1227.522,160.462,-52.637,-177.813,5.798,148.374
C01144=1227.518,160.711,-52.659,-177.811,5.799,148.373
C01145=1227.513,160.960,-52.681,-177.808,5.801,148.373
C01146=1227.508,161.209,-52.702,-177.806,5.802,148.372
C01147=1227.504,161.458,-52.724,-177.803,5.803,148.372
C01148=1227.499,161.708,-52.745,-177.801,5.804,148.371
C01149=1227.494,161.956,-52.767,-177.798,5.806,148.371
C01150=1227.490,162.205,-52.789,-177.795,5.807,148.370
C01151=1227.485,162.454,-52.811,-177.793,5.809,148.370
C01152=1227.481,162.703,-52.833,-177.791,5.810,148.369
C01153=1227.476,162.952,-52.855,-177.788,5.811,148.369
C01154=1227.470,163.201,-52.877,-177.785,5.812,148.368
C01155=1227.466,163.450,-52.899,-177.782,5.814,148.368
C01156=1227.461,163.699,-52.921,-177.780,5.815,148.367
C01157=1227.457,163.948,-52.943,-177.778,5.816,148.367
C01158=1227.452,164.197,-52.964,-177.774,5.818,148.367
C01159=1227.448,164.446,-52.986,-177.772,5.819,148.366
C01160=1227.443,164.695,-53.008,-177.770,5.821,148.366
C01161=1227.439,164.944,-53.030,-177.767,5.821,148.365
C01162=1227.434,165.193,-53.052,-177.764,5.823,148.365
C01163=1227.429,165.442,-53.074,-177.762,5.824,148.364
C01164=1227.424,165.691,-53.096,-177.760,5.826,148.364
C01165=1227.420,165.941,-53.118,-177.757,5.827,148.363
C01166=1227.415,166.189,-53.140,-177.754,5.829,148.363
C01167=1227.410,166.439,-53.162,-177.752,5.830,148.363
C01168=1227.406,166.687,-53.184,-177.749,5.831,148.362
C01169=1227.401,166.937,-53.206,-177.747,5.833,148.362
C01170=1227.396,167.185,-53.227,-177.744,5.834,148.361
C01171=1227.391,167.435,-53.250,-177.741,5.835,148.361
C01172=1227.387,167.683,-53.272,-177.739,5.836,148.360
C01173=1227.383,167.932,-53.294,-177.737,5.838,148.360
C01174=1227.378,168.181,-53.316,-177.734,5.839,148.359
C01175=1227.373,168.430,-53.338,-177.731,5.841,148.359
C01176=1227.368,168.679,-53.360,-177.729,5.842,148.359
C01177=1227.364,168.929,-53.382,-177.726,5.843,148.358
C01178=1227.359,169.177,-53.404,-177.723,5.845,148.358
C01179=1227.355,169.426,-53.427,-177.721,5.846,148.357
C01180=1227.349,169.675,-53.449,-177.719,5.848,148.357
C01181=1227.345,169.924,-53.471,-177.716,5.848,148.356
C01182=1227.340,170.173,-53.493,-177.713,5.850,148.356
C01183=1227.336,170.422,-53.516,-177.711,5.851,148.356
C01184=1227.330,170.670,-53.538,-177.708,5.853,148.355
C01185=1227.326,170.920,-53.560,-177.705,5.855,148.355
C01186=1227.322,171.169,-53.582,-177.703,5.856,148.354
C01187=1227.317,171.417,-53.604,-177.700,5.857,148.354
C01188=1227.312,171.667,-53.627,-177.698,5.858,148.353
C01189=1227.307,171.915,-53.649,-177.696,5.860,148.353
C01190=1227.303,172.165,-53.671,-177.693,5.861,148.353
C01191=1227.298,172.413,-53.694,-177.690,5.862,148.352
C01192=1227.294,172.662,-53.716,-177.688,5.864,148.352
C01193=1227.289,172.912,-53.738,-177.686,5.865,148.351
C01194=1227.284,173.160,-53.761,-177.682,5.867,148.351
C01195=1227.280,173.410,-53.783,-177.680,5.868,148.350
C01196=1227.275,173.658,-53.805,-177.678,5.870,148.350
C01197=1227.270,173.907,-53.828,-177.675,5.872,148.350
C01198=1227.266,174.157,-53.850,-177.672,5.872,148.349
C01199=1227.261,174.405,-53.872,-177.670,5.874,148.349
C01200=1227.256,174.654,-53.895,-177.668,5.875,148.348
C01201=1227.252,174.904,-53.917,-177.665,5.877,148.348
C01202=1227.247,175.152,-53.940,-177.662,5.878,148.347
C01203=1227.243,175.401,-53.962,-177.660,5.879,148.347
C01204=1227.239,175.650,-53.985,-177.657,5.881,148.346
C01205=1227.233,175.899,-54.007,-177.655,5.882,148.346
C01206=1227.229,176.148,-54.030,-177.652,5.884,148.346
C01207=1227.223,176.397,-54.052,-177.649,5.886,148.345
C01208=1227.219,176.646,-54.074,-177.647,5.887,148.345
C01209=1227.214,176.895,-54.098,-177.644,5.888,148.344
C01210=1227.210,177.144,-54.119,-177.641,5.890,148.344
C01211=1227.206,177.392,-54.142,-177.639,5.891,148.343
C01212=1227.201,177.641,-54.165,-177.637,5.893,148.343
C01213=1227.197,177.891,-54.188,-177.634,5.893,148.342
C01214=1227.191,178.139,-54.211,-177.631,5.895,148.342
C01215=1227.187,178.388,-54.233,-177.629,5.897,148.342
C01216=1227.182,178.637,-54.256,-177.627,5.898,148.341
C01217=1227.177,178.886,-54.278,-177.623,5.900,148.341
C01218=1227.173,179.135,-54.301,-177.621,5.901,148.340
C01219=1227.169,179.384,-54.323,-177.619,5.902,148.340
C01220=1227.163,179.633,-54.346,-177.616,5.904,148.340
C01221=1227.159,179.881,-54.369,-177.614,5.905,148.339
C01222=1227.154,180.131,-54.391,-177.611,5.907,148.339
C01223=1227.150,180.380,-54.414,-177.608,5.909,148.338
C01224=1227.145,180.628,-54.437,-177.606,5.910,148.338
C01225=1227.141,180.877,-54.459,-177.603,5.911,148.338
C01226=1227.136,181.127,-54.483,-177.600,5.913,148.337
C01227=1227.131,181.376,-54.506,-177.598,5.914,148.337
C01228=1227.126,181.624,-54.528,-177.596,5.916,148.336
C01229=1227.122,181.873,-54.551,-177.593,5.918,148.336
C01230=1227.118,182.122,-54.574,-177.590,5.918,148.335
C01231=1227.113,182.372,-54.596,-177.588,5.920,148.335
C01232=1227.108,182.620,-54.619,-177.586,5.921,148.335
C01233=1227.104,182.869,-54.642,-177.583,5.923,148.334
C01234=1227.099,183.118,-54.666,-177.580,5.925,148.334
C01235=1227.095,183.367,-54.688,-177.578,5.926,148.333
C01236=1227.089,183.615,-54.711,-177.575,5.927,148.333
C01237=1227.085,183.864,-54.733,-177.572,5.929,148.333
C01238=1227.081,184.113,-54.757,-177.570,5.930,148.332
C01239=1227.076,184.363,-54.779,-177.567,5.932,148.332
C01240=1227.072,184.611,-54.802,-177.565,5.934,148.331
C01241=1227.066,184.860,-54.825,-177.563,5.935,148.331
C01242=1227.062,185.109,-54.848,-177.560,5.936,148.331
C01243=1227.057,185.378,-54.873,-177.557,5.938,148.330
C01244=1227.052,185.648,-54.898,-177.554,5.940,148.330
C01245=1227.046,185.918,-54.923,-177.551,5.942,148.329
C01246=1227.042,186.187,-54.947,-177.548,5.943,148.329
C01247=1227.037,186.436,-54.971,-177.546,5.944,148.328
C01248=1227.032,186.685,-54.994,-177.544,5.946,148.328
C01249=1227.028,186.934,-55.017,-177.541,5.948,148.328
C01250=1227.024,187.183,-55.040,-177.538,5.948,148.327
C01251=1227.019,187.432,-55.064,-177.536,5.950,148.327
C01252=1227.014,187.680,-55.087,-177.533,5.952,148.326
C01253=1227.010,187.929,-55.109,-177.531,5.953,148.326
C01254=1227.005,188.178,-55.133,-177.528,5.955,148.326
C01255=1227.000,188.427,-55.156,-177.526,5.957,148.325
C01256=1226.995,188.677,-55.179,-177.523,5.958,148.325
C01257=1226.991,188.926,-55.201,-177.520,5.959,148.324
C01258=1226.987,189.175,-55.225,-177.518,5.961,148.324
C01259=1226.982,189.424,-55.248,-177.515,5.963,148.324
C01260=1226.977,189.672,-55.271,-177.513,5.964,148.323
C01261=1226.972,189.921,-55.295,-177.510,5.966,148.323
C01262=1226.968,190.169,-55.318,-177.507,5.967,148.322
C01263=1226.964,190.418,-55.341,-177.505,5.968,148.322
C01264=1226.959,190.667,-55.365,-177.503,5.970,148.322
C01265=1226.954,190.916,-55.388,-177.500,5.972,148.321
C01266=1226.950,191.165,-55.411,-177.497,5.974,148.321
C01267=1226.945,191.414,-55.435,-177.495,5.975,148.320
C01268=1226.941,191.663,-55.458,-177.492,5.977,148.320
C01269=1226.936,191.912,-55.481,-177.489,5.978,148.320
C01270=1226.932,192.161,-55.504,-177.487,5.979,148.319
C01271=1226.926,192.409,-55.527,-177.485,5.981,148.319
C01272=1226.922,192.658,-55.551,-177.482,5.983,148.319
C01273=1226.917,192.907,-55.575,-177.480,5.984,148.318
C01274=1226.912,193.156,-55.598,-177.477,5.986,148.318
C01275=1226.908,193.405,-55.621,-177.474,5.987,148.317
C01276=1226.904,193.654,-55.644,-177.472,5.989,148.317
C01277=1226.899,193.903,-55.668,-177.470,5.990,148.317
C01278=1226.894,194.152,-55.691,-177.467,5.992,148.316
C01279=1226.890,194.400,-55.715,-177.464,5.994,148.316
C01280=1226.885,194.649,-55.738,-177.461,5.996,148.315
C01281=1226.881,194.898,-55.762,-177.459,5.997,148.315
C01282=1226.876,195.147,-55.785,-177.456,5.998,148.315
C01283=1226.871,195.396,-55.809,-177.454,6.000,148.314
C01284=1226.867,195.645,-55.832,-177.451,6.002,148.314
C01285=1226.862,195.894,-55.856,-177.449,6.003,148.314
C01286=1226.857,196.143,-55.879,-177.446,6.005,148.313
C01287=1226.853,196.391,-55.903,-177.443,6.006,148.313
C01288=1226.848,196.640,-55.927,-177.441,6.007,148.312
C01289=1226.844,196.889,-55.950,-177.439,6.009,148.312
C01290=1226.839,197.138,-55.974,-177.436,6.011,148.312
C01291=1226.834,197.387,-55.997,-177.433,6.013,148.311
C01292=1226.830,197.636,-56.021,-177.431,6.014,148.311
C01293=1226.825,197.884,-56.045,-177.429,6.016,148.310
C01294=1226.821,198.133,-56.068,-177.425,6.017,148.310
C01295=1226.816,198.382,-56.092,-177.423,6.019,148.310
C01296=1226.812,198.631,-56.116,-177.421,6.020,148.309
C01297=1226.807,198.880,-56.139,-177.418,6.022,148.309
C01298=1226.803,199.128,-56.163,-177.415,6.024,148.309
C01299=1226.798,199.377,-56.186,-177.413,6.026,148.308
C01300=1226.793,199.626,-56.210,-177.410,6.028,148.308
C01301=1226.789,199.874,-56.234,-177.408,6.029,148.307
C01302=1226.785,200.124,-56.258,-177.405,6.030,148.307
C01303=1226.780,200.373,-56.282,-177.402,6.032,148.307
C01304=1226.775,200.622,-56.306,-177.400,6.034,148.306
C01305=1226.770,200.870,-56.330,-177.398,6.035,148.306
C01306=1226.766,201.119,-56.353,-177.395,6.037,148.305
C01307=1226.761,201.368,-56.377,-177.392,6.039,148.305
C01308=1226.757,201.617,-56.401,-177.390,6.041,148.305
C01309=1226.752,201.865,-56.425,-177.388,6.042,148.304
C01310=1226.747,202.114,-56.448,-177.385,6.043,148.304
C01311=1226.743,202.363,-56.472,-177.382,6.045,148.304
C01312=1226.738,202.612,-56.496,-177.379,6.047,148.303
C01313=1226.734,202.861,-56.520,-177.377,6.049,148.303
C01314=1226.729,203.110,-56.544,-177.374,6.050,148.302
C01315=1226.725,203.359,-56.568,-177.372,6.051,148.302
C01316=1226.720,203.607,-56.592,-177.369,6.053,148.302
C01317=1226.716,203.856,-56.615,-177.367,6.055,148.301
C01318=1226.711,204.105,-56.640,-177.364,6.057,148.301
C01319=1226.706,204.353,-56.664,-177.362,6.058,148.301
C01320=1226.702,204.603,-56.688,-177.359,6.060,148.300
C01321=1226.698,204.851,-56.712,-177.357,6.062,148.300
C01322=1226.693,205.100,-56.736,-177.353,6.063,148.300
C01323=1226.688,205.349,-56.760,-177.351,6.065,148.299
C01324=1226.683,205.598,-56.784,-177.349,6.066,148.299
C01325=1226.679,205.846,-56.808,-177.346,6.068,148.298
C01326=1226.675,206.096,-56.832,-177.343,6.070,148.298
C01327=1226.670,206.344,-56.856,-177.341,6.072,148.298
C01328=1226.665,206.593,-56.880,-177.338,6.074,148.297
C01329=1226.661,206.842,-56.904,-177.336,6.075,148.297
C01330=1226.656,207.090,-56.928,-177.333,6.076,148.297
C01331=1226.651,207.339,-56.953,-177.331,6.078,148.296
C01332=1226.647,207.588,-56.977,-177.328,6.080,148.296
C01333=1226.643,207.837,-57.000,-177.326,6.082,148.296
C01334=1226.638,208.086,-57.025,-177.323,6.083,148.295
C01335=1226.633,208.334,-57.049,-177.321,6.085,148.295
C01336=1226.629,208.583,-57.073,-177.318,6.086,148.294
C01337=1226.624,208.832,-57.098,-177.315,6.088,148.294
C01338=1226.620,209.081,-57.122,-177.312,6.090,148.294
C01339=1226.615,209.330,-57.146,-177.310,6.092,148.293
C01340=1226.610,209.578,-57.170,-177.308,6.093,148.293
C01341=1226.606,209.827,-57.195,-177.305,6.095,148.293
C01342=1226.602,210.076,-57.219,-177.302,6.097,148.292
C01343=1226.597,210.325,-57.244,-177.300,6.099,148.292
C01344=1226.592,210.573,-57.268,-177.297,6.100,148.292
C01345=1226.588,210.822,-57.293,-177.295,6.102,148.291
C01346=1226.583,211.071,-57.317,-177.292,6.103,148.291
C01347=1226.578,211.342,-57.343,-177.290,6.105,148.291
C01348=1226.573,211.612,-57.369,-177.286,6.108,148.290
C01349=1226.568,211.882,-57.396,-177.284,6.109,148.290
C01350=1226.564,212.152,-57.423,-177.281,6.111,148.290
C01351=1226.559,212.401,-57.447,-177.278,6.113,148.289
C01352=1226.554,212.650,-57.471,-177.276,6.114,148.289
C01353=1226.550,212.899,-57.495,-177.274,6.116,148.289
C01354=1226.545,213.148,-57.520,-177.271,6.118,148.288
C01355=1226.541,213.396,-57.544,-177.268,6.120,148.288
C01356=1226.536,213.645,-57.569,-177.266,6.122,148.288
C01357=1226.532,213.894,-57.594,-177.263,6.123,148.287
C01358=1226.527,214.142,-57.618,-177.260,6.125,148.287
C01359=1226.523,214.391,-57.642,-177.258,6.126,148.286
C01360=1226.518,214.640,-57.667,-177.256,6.128,148.286
C01361=1226.514,214.889,-57.691,-177.253,6.130,148.286
C01362=1226.508,215.137,-57.716,-177.250,6.132,148.285
C01363=1226.505,215.386,-57.741,-177.248,6.134,148.285
C01364=1226.500,215.635,-57.765,-177.245,6.136,148.285
C01365=1226.495,215.884,-57.789,-177.243,6.137,148.285
C01366=1226.491,216.133,-57.814,-177.241,6.139,148.284
C01367=1226.486,216.381,-57.838,-177.238,6.140,148.284
C01368=1226.481,216.630,-57.864,-177.235,6.142,148.283
C01369=1226.477,216.879,-57.889,-177.233,6.144,148.283
C01370=1226.472,217.127,-57.913,-177.230,6.146,148.283
C01371=1226.468,217.377,-57.938,-177.227,6.148,148.282
C01372=1226.464,217.625,-57.962,-177.225,6.150,148.282
C01373=1226.459,217.873,-57.987,-177.222,6.152,148.282
C01374=1226.454,218.123,-58.012,-177.219,6.153,148.281
C01375=1226.450,218.371,-58.037,-177.217,6.154,148.281
C01376=1226.445,218.621,-58.062,-177.215,6.156,148.281
C01377=1226.441,218.869,-58.086,-177.212,6.158,148.280
C01378=1226.436,219.117,-58.111,-177.210,6.160,148.280
C01379=1226.432,219.367,-58.136,-177.207,6.162,148.280
C01380=1226.427,219.615,-58.160,-177.204,6.164,148.279
C01381=1226.423,219.864,-58.186,-177.202,6.166,148.279
C01382=1226.418,220.112,-58.211,-177.199,6.167,148.279
C01383=1226.413,220.361,-58.235,-177.197,6.168,148.278
C01384=1226.409,220.610,-58.260,-177.194,6.170,148.278
C01385=1226.404,220.858,-58.285,-177.192,6.172,148.278
C01386=1226.400,221.108,-58.310,-177.189,6.174,148.277
C01387=1226.395,221.356,-58.335,-177.186,6.176,148.277
C01388=1226.391,221.605,-58.360,-177.184,6.178,148.277
C01389=1226.386,221.853,-58.384,-177.181,6.180,148.277
C01390=1226.382,222.102,-58.410,-177.179,6.182,148.276
C01391=1226.377,222.351,-58.434,-177.176,6.183,148.276
C01392=1226.373,222.599,-58.459,-177.173,6.185,148.276
C01393=1226.368,222.848,-58.484,-177.171,6.186,148.275
C01394=1226.363,223.097,-58.509,-177.169,6.188,148.275
C01395=1226.359,223.346,-58.535,-177.166,6.190,148.275
C01396=1226.355,223.594,-58.559,-177.163,6.192,148.274
C01397=1226.351,223.843,-58.584,-177.161,6.194,148.274
C01398=1226.345,224.092,-58.609,-177.158,6.196,148.274
C01399=1226.341,224.341,-58.635,-177.155,6.197,148.273
C01400=1226.337,224.589,-58.659,-177.153,6.199,148.273
C01401=1226.333,224.838,-58.685,-177.150,6.201,148.273
C01402=1226.327,225.086,-58.709,-177.148,6.203,148.272
C01403=1226.323,225.335,-58.735,-177.146,6.204,148.272
C01404=1226.318,225.584,-58.760,-177.143,6.206,148.272
C01405=1226.314,225.833,-58.786,-177.141,6.208,148.271
C01406=1226.309,226.081,-58.810,-177.138,6.210,148.271
C01407=1226.305,226.330,-58.835,-177.136,6.212,148.271
C01408=1226.301,226.579,-58.861,-177.133,6.214,148.270
C01409=1226.296,226.828,-58.886,-177.130,6.216,148.270
C01410=1226.292,227.076,-58.912,-177.128,6.218,148.270
C01411=1226.286,227.325,-58.936,-177.125,6.219,148.270
C01412=1226.283,227.574,-58.961,-177.122,6.221,148.269
C01413=1226.278,227.822,-58.987,-177.120,6.223,148.269
C01414=1226.274,228.071,-59.012,-177.117,6.225,148.269
C01415=1226.269,228.319,-59.037,-177.115,6.226,148.268
C01416=1226.265,228.568,-59.063,-177.112,6.228,148.268
C01417=1226.260,228.817,-59.088,-177.110,6.230,148.268
C01418=1226.255,229.066,-59.113,-177.108,6.232,148.267
C01419=1226.251,229.314,-59.139,-177.105,6.234,148.267
C01420=1226.246,229.563,-59.164,-177.102,6.236,148.267
C01421=1226.242,229.812,-59.190,-177.100,6.238,148.266
C01422=1226.237,230.060,-59.215,-177.097,6.239,148.266
C01423=1226.233,230.308,-59.240,-177.095,6.241,148.266
C01424=1226.229,230.558,-59.265,-177.092,6.243,148.266
C01425=1226.224,230.806,-59.291,-177.089,6.245,148.265
C01426=1226.220,231.055,-59.316,-177.087,6.247,148.265
C01427=1226.216,231.304,-59.342,-177.084,6.249,148.265
C01428=1226.210,231.552,-59.367,-177.082,6.251,148.264
C01429=1226.206,231.801,-59.392,-177.080,6.252,148.264
C01430=1226.201,232.049,-59.418,-177.077,6.254,148.264
C01431=1226.197,232.298,-59.444,-177.075,6.256,148.263
C01432=1226.193,232.547,-59.469,-177.072,6.258,148.263
C01433=1226.188,232.795,-59.495,-177.069,6.259,148.263
C01434=1226.184,233.044,-59.520,-177.067,6.261,148.262
C01435=1226.179,233.293,-59.545,-177.064,6.263,148.262
C01436=1226.175,233.541,-59.571,-177.062,6.265,148.262
C01437=1226.170,233.790,-59.597,-177.059,6.267,148.262
C01438=1226.165,234.039,-59.623,-177.057,6.269,148.261
C01439=1226.160,234.287,-59.648,-177.054,6.271,148.261
C01440=1226.156,234.536,-59.674,-177.052,6.273,148.261
C01441=1226.152,234.785,-59.700,-177.049,6.275,148.260
C01442=1226.147,235.033,-59.725,-177.046,6.277,148.260
C01443=1226.143,235.282,-59.751,-177.044,6.278,148.260
C01444=1226.139,235.531,-59.777,-177.042,6.281,148.260
C01445=1226.134,235.779,-59.802,-177.039,6.283,148.259
C01446=1226.130,236.027,-59.828,-177.036,6.284,148.259
C01447=1226.125,236.276,-59.854,-177.034,6.286,148.259
C01448=1226.121,236.525,-59.880,-177.031,6.288,148.258
C01449=1226.116,236.774,-59.905,-177.028,6.290,148.258
C01450=1226.111,237.022,-59.931,-177.026,6.291,148.258
C01451=1226.107,237.294,-59.959,-177.023,6.294,148.258
C01452=1226.101,237.565,-59.987,-177.021,6.296,148.257
C01453=1226.097,237.837,-60.016,-177.018,6.298,148.257
C01454=1226.092,238.108,-60.043,-177.015,6.299,148.257
C01455=1226.088,238.357,-60.069,-177.013,6.302,148.256
C01456=1226.083,238.606,-60.095,-177.011,6.303,148.256
C01457=1226.079,238.854,-60.122,-177.008,6.305,148.256
C01458=1226.074,239.102,-60.147,-177.005,6.307,148.256
C01459=1226.070,239.351,-60.173,-177.003,6.309,148.255
C01460=1226.065,239.600,-60.199,-177.000,6.311,148.255
C01461=1226.060,239.849,-60.225,-176.998,6.313,148.255
C01462=1226.056,240.097,-60.250,-176.995,6.315,148.254
C01463=1226.051,240.346,-60.276,-176.993,6.317,148.254
C01464=1226.048,240.594,-60.303,-176.990,6.319,148.254
C01465=1226.043,240.843,-60.328,-176.988,6.321,148.254
C01466=1226.038,241.092,-60.355,-176.985,6.323,148.253
C01467=1226.033,241.340,-60.380,-176.983,6.325,148.253
C01468=1226.030,241.588,-60.407,-176.980,6.327,148.253
C01469=1226.025,241.837,-60.433,-176.978,6.328,148.253
C01470=1226.020,242.086,-60.459,-176.975,6.330,148.252
C01471=1226.016,242.335,-60.484,-176.972,6.332,148.252
C01472=1226.012,242.582,-60.511,-176.970,6.334,148.252
C01473=1226.007,242.831,-60.537,-176.968,6.336,148.251
C01474=1226.002,243.080,-60.563,-176.965,6.338,148.251
C01475=1225.999,243.328,-60.589,-176.962,6.340,148.251
C01476=1225.994,243.578,-60.615,-176.960,6.342,148.251
C01477=1225.989,243.826,-60.641,-176.958,6.344,148.250
C01478=1225.985,244.074,-60.667,-176.955,6.346,148.250
C01479=1225.980,244.323,-60.694,-176.952,6.348,148.250
C01480=1225.976,244.572,-60.719,-176.950,6.350,148.250
C01481=1225.971,244.820,-60.746,-176.948,6.352,148.249
C01482=1225.967,245.069,-60.772,-176.945,6.354,148.249
C01483=1225.963,245.318,-60.798,-176.942,6.356,148.249
C01484=1225.958,245.566,-60.825,-176.940,6.358,148.248
C01485=1225.953,245.814,-60.850,-176.937,6.359,148.248
C01486=1225.948,246.063,-60.877,-176.935,6.362,148.248
C01487=1225.944,246.312,-60.903,-176.932,6.364,148.248
C01488=1225.940,246.560,-60.930,-176.930,6.365,148.247
C01489=1225.935,246.809,-60.956,-176.927,6.367,148.247
C01490=1225.931,247.057,-60.983,-176.925,6.369,148.247
C01491=1225.926,247.306,-61.009,-176.922,6.371,148.247
C01492=1225.922,247.555,-61.035,-176.920,6.373,148.246
C01493=1225.918,247.804,-61.062,-176.917,6.375,148.246
C01494=1225.914,248.052,-61.088,-176.915,6.377,148.246
C01495=1225.908,248.300,-61.114,-176.912,6.379,148.246
C01496=1225.904,248.548,-61.141,-176.910,6.381,148.245
C01497=1225.900,248.797,-61.166,-176.907,6.384,148.245
C01498=1225.895,249.046,-61.193,-176.905,6.386,148.245
C01499=1225.891,249.295,-61.219,-176.902,6.388,148.245
C01500=1225.886,249.543,-61.246,-176.899,6.390,148.244
C01501=1225.882,249.792,-61.273,-176.897,6.392,148.244
C01502=1225.877,250.040,-61.299,-176.895,6.394,148.244
C01503=1225.873,250.289,-61.326,-176.892,6.396,148.244
C01504=1225.869,250.538,-61.352,-176.889,6.398,148.243
C01505=1225.864,250.786,-61.379,-176.887,6.399,148.243
C01506=1225.860,251.034,-61.405,-176.885,6.402,148.243
C01507=1225.855,251.283,-61.432,-176.882,6.404,148.243
C01508=1225.851,251.532,-61.458,-176.879,6.405,148.242
C01509=1225.846,251.780,-61.485,-176.877,6.407,148.242
C01510=1225.843,252.028,-61.512,-176.875,6.410,148.242
C01511=1225.838,252.277,-61.538,-176.872,6.411,148.242
C01512=1225.833,252.526,-61.565,-176.869,6.413,148.241
C01513=1225.829,252.774,-61.592,-176.867,6.415,148.241
C01514=1225.824,253.023,-61.618,-176.865,6.417,148.241
C01515=1225.819,253.272,-61.645,-176.862,6.419,148.241
C01516=1225.815,253.520,-61.671,-176.860,6.421,148.240
C01517=1225.811,253.768,-61.699,-176.857,6.423,148.240
C01518=1225.807,254.017,-61.725,-176.854,6.426,148.240
C01519=1225.802,254.266,-61.751,-176.852,6.428,148.240
C01520=1225.797,254.514,-61.778,-176.849,6.430,148.240
C01521=1225.793,254.762,-61.805,-176.847,6.432,148.239
C01522=1225.789,255.011,-61.832,-176.844,6.434,148.239
C01523=1225.784,255.259,-61.859,-176.842,6.436,148.239
C01524=1225.780,255.508,-61.885,-176.840,6.438,148.239
C01525=1225.775,255.757,-61.912,-176.837,6.440,148.238
C01526=1225.771,256.005,-61.939,-176.835,6.442,148.238
C01527=1225.766,256.254,-61.966,-176.832,6.444,148.238
C01528=1225.762,256.502,-61.992,-176.830,6.446,148.238
C01529=1225.757,256.750,-62.019,-176.827,6.448,148.237
C01530=1225.753,257.000,-62.047,-176.825,6.450,148.237
C01531=1225.749,257.248,-62.073,-176.822,6.452,148.237
C01532=1225.745,257.496,-62.100,-176.819,6.455,148.237
C01533=1225.740,257.745,-62.127,-176.817,6.457,148.237
C01534=1225.735,257.993,-62.155,-176.814,6.459,148.236
C01535=1225.731,258.241,-62.181,-176.812,6.460,148.236
C01536=1225.727,258.490,-62.208,-176.810,6.463,148.236
C01537=1225.722,258.738,-62.235,-176.807,6.465,148.236
C01538=1225.717,258.987,-62.262,-176.804,6.466,148.235
C01539=1225.713,259.235,-62.289,-176.802,6.469,148.235
C01540=1225.709,259.484,-62.316,-176.800,6.471,148.235
C01541=1225.705,259.733,-62.343,-176.798,6.473,148.235
C01542=1225.700,259.981,-62.370,-176.795,6.475,148.235
C01543=1225.696,260.230,-62.397,-176.792,6.477,148.234
C01544=1225.691,260.478,-62.424,-176.790,6.480,148.234
C01545=1225.686,260.727,-62.451,-176.787,6.481,148.234
C01546=1225.682,260.975,-62.478,-176.784,6.483,148.234
C01547=1225.678,261.224,-62.505,-176.782,6.486,148.234
C01548=1225.674,261.473,-62.532,-176.780,6.487,148.233
C01549=1225.669,261.721,-62.560,-176.777,6.489,148.233
C01550=1225.665,261.969,-62.587,-176.775,6.492,148.233
C01551=1225.660,262.217,-62.614,-176.772,6.493,148.233
C01552=1225.655,262.466,-62.641,-176.770,6.496,148.233
C01553=1225.652,262.715,-62.668,-176.767,6.498,148.232
C01554=1225.647,262.963,-62.695,-176.764,6.500,148.232
C01555=1225.642,263.236,-62.725,-176.762,6.502,148.232
C01556=1225.637,263.508,-62.755,-176.759,6.505,148.232
C01557=1225.632,263.781,-62.786,-176.757,6.507,148.231
C01558=1225.628,264.053,-62.815,-176.753,6.510,148.231
C01559=1225.623,264.302,-62.842,-176.751,6.512,148.231
C01560=1225.619,264.551,-62.870,-176.749,6.514,148.231
C01561=1225.615,264.799,-62.897,-176.746,6.516,148.230
C01562=1225.610,265.047,-62.925,-176.744,6.518,148.230
C01563=1225.605,265.296,-62.952,-176.741,6.520,148.230
C01564=1225.601,265.545,-62.979,-176.739,6.522,148.230
C01565=1225.597,265.793,-63.007,-176.737,6.524,148.230
C01566=1225.592,266.041,-63.034,-176.733,6.527,148.229
C01567=1225.588,266.290,-63.061,-176.731,6.529,148.229
C01568=1225.584,266.538,-63.089,-176.729,6.531,148.229
C01569=1225.579,266.787,-63.116,-176.727,6.533,148.229
C01570=1225.575,267.035,-63.144,-176.724,6.535,148.229
C01571=1225.570,267.283,-63.171,-176.722,6.537,148.229
C01572=1225.566,267.533,-63.198,-176.719,6.539,148.228
C01573=1225.562,267.780,-63.226,-176.716,6.542,148.228
C01574=1225.557,268.029,-63.253,-176.714,6.544,148.228
C01575=1225.553,268.277,-63.281,-176.711,6.546,148.228
C01576=1225.549,268.526,-63.308,-176.709,6.548,148.228
C01577=1225.544,268.774,-63.336,-176.707,6.550,148.227
C01578=1225.539,269.023,-63.364,-176.705,6.552,148.227
C01579=1225.535,269.272,-63.391,-176.702,6.554,148.227
C01580=1225.531,269.520,-63.419,-176.699,6.557,148.227
C01581=1225.526,269.768,-63.446,-176.697,6.559,148.227
C01582=1225.522,270.016,-63.474,-176.694,6.561,148.226
C01583=1225.518,270.265,-63.502,-176.692,6.563,148.226
C01584=1225.513,270.513,-63.529,-176.689,6.565,148.226
C01585=1225.509,270.761,-63.557,-176.687,6.567,148.226
C01586=1225.504,271.011,-63.585,-176.684,6.570,148.226
C01587=1225.500,271.258,-63.613,-176.682,6.572,148.225
C01588=1225.495,271.507,-63.640,-176.679,6.574,148.225
C01589=1225.491,271.755,-63.668,-176.677,6.576,148.225
C01590=1225.487,272.004,-63.695,-176.675,6.578,148.225
C01591=1225.482,272.252,-63.723,-176.673,6.580,148.225
C01592=1225.478,272.501,-63.751,-176.669,6.583,148.225
C01593=1225.473,272.749,-63.779,-176.667,6.585,148.224
C01594=1225.469,272.998,-63.807,-176.665,6.587,148.224
C01595=1225.465,273.246,-63.834,-176.663,6.589,148.224
C01596=1225.460,273.494,-63.862,-176.660,6.591,148.224
C01597=1225.456,273.743,-63.890,-176.657,6.594,148.224
C01598=1225.451,273.991,-63.918,-176.655,6.596,148.223
C01599=1225.447,274.239,-63.945,-176.653,6.598,148.223
C01600=1225.443,274.488,-63.973,-176.650,6.600,148.223
C01601=1225.438,274.736,-64.002,-176.648,6.602,148.223
C01602=1225.434,274.985,-64.030,-176.645,6.604,148.223
C01603=1225.430,275.233,-64.057,-176.643,6.607,148.223
C01604=1225.425,275.481,-64.085,-176.640,6.609,148.222
C01605=1225.421,275.730,-64.113,-176.638,6.611,148.222
C01606=1225.416,275.978,-64.141,-176.635,6.613,148.222
C01607=1225.413,276.226,-64.169,-176.633,6.615,148.222
C01608=1225.407,276.475,-64.197,-176.630,6.618,148.222
C01609=1225.404,276.724,-64.225,-176.628,6.620,148.222
C01610=1225.399,276.972,-64.253,-176.625,6.622,148.221
C01611=1225.394,277.220,-64.281,-176.623,6.625,148.221
C01612=1225.390,277.469,-64.309,-176.621,6.626,148.221
C01613=1225.386,277.716,-64.337,-176.618,6.629,148.221
C01614=1225.381,277.966,-64.365,-176.615,6.631,148.221
C01615=1225.377,278.214,-64.393,-176.613,6.634,148.221
C01616=1225.373,278.462,-64.421,-176.611,6.636,148.221
C01617=1225.368,278.711,-64.449,-176.608,6.639,148.220
C01618=1225.364,278.959,-64.478,-176.606,6.641,148.220
C01619=1225.360,279.207,-64.505,-176.603,6.643,148.220
C01620=1225.355,279.456,-64.534,-176.601,6.645,148.220
C01621=1225.351,279.704,-64.562,-176.598,6.647,148.220
C01622=1225.347,279.953,-64.591,-176.596,6.650,148.220
C01623=1225.342,280.201,-64.618,-176.593,6.652,148.219
C01624=1225.338,280.449,-64.647,-176.591,6.654,148.219
C01625=1225.333,280.697,-64.675,-176.589,6.656,148.219
C01626=1225.330,280.946,-64.703,-176.586,6.658,148.219
C01627=1225.325,281.194,-64.731,-176.584,6.661,148.219
C01628=1225.321,281.443,-64.760,-176.581,6.663,148.219
C01629=1225.316,281.691,-64.788,-176.579,6.665,148.218
C01630=1225.312,281.939,-64.816,-176.577,6.667,148.218
C01631=1225.307,282.188,-64.844,-176.574,6.670,148.218
C01632=1225.303,282.436,-64.873,-176.572,6.672,148.218
C01633=1225.298,282.684,-64.901,-176.569,6.674,148.218
C01634=1225.294,282.933,-64.929,-176.567,6.676,148.218
C01635=1225.290,283.182,-64.958,-176.564,6.679,148.218
C01636=1225.286,283.429,-64.986,-176.562,6.681,148.217
C01637=1225.281,283.678,-65.015,-176.560,6.684,148.217
C01638=1225.277,283.926,-65.043,-176.557,6.685,148.217
C01639=1225.272,284.175,-65.072,-176.554,6.688,148.217
C01640=1225.268,284.423,-65.099,-176.552,6.691,148.217
C01641=1225.264,284.671,-65.128,-176.550,6.693,148.217
C01642=1225.259,284.919,-65.157,-176.547,6.695,148.217
C01643=1225.255,285.168,-65.185,-176.545,6.698,148.217
C01644=1225.251,285.416,-65.214,-176.542,6.700,148.216
C01645=1225.246,285.664,-65.242,-176.540,6.702,148.216
C01646=1225.242,285.913,-65.271,-176.538,6.704,148.216
C01647=1225.238,286.160,-65.299,-176.535,6.707,148.216
C01648=1225.233,286.409,-65.328,-176.533,6.709,148.216
C01649=1225.229,286.658,-65.357,-176.531,6.711,148.216
C01650=1225.225,286.906,-65.385,-176.528,6.713,148.216
C01651=1225.220,287.154,-65.414,-176.525,6.716,148.216
C01652=1225.216,287.403,-65.443,-176.523,6.718,148.215
C01653=1225.212,287.651,-65.471,-176.521,6.720,148.215
C01654=1225.207,287.899,-65.500,-176.519,6.723,148.215
C01655=1225.202,288.148,-65.528,-176.516,6.726,148.215
C01656=1225.199,288.396,-65.557,-176.513,6.728,148.215
C01657=1225.194,288.644,-65.586,-176.511,6.730,148.215
C01658=1225.189,288.893,-65.614,-176.509,6.732,148.215
C01659=1225.185,289.166,-65.646,-176.506,6.735,148.214
C01660=1225.180,289.440,-65.677,-176.503,6.738,148.214
C01661=1225.176,289.715,-65.709,-176.501,6.740,148.214
C01662=1225.171,289.989,-65.741,-176.498,6.743,148.214
C01663=1225.166,290.237,-65.770,-176.496,6.745,148.214
C01664=1225.162,290.486,-65.799,-176.493,6.747,148.214
C01665=1225.157,290.734,-65.828,-176.491,6.750,148.214
C01666=1225.154,290.982,-65.856,-176.488,6.752,148.214
C01667=1225.149,291.230,-65.885,-176.486,6.754,148.213
C01668=1225.144,291.479,-65.914,-176.483,6.757,148.213
C01669=1225.140,291.727,-65.943,-176.481,6.759,148.213
C01670=1225.136,291.975,-65.971,-176.479,6.761,148.213
C01671=1225.132,292.223,-66.001,-176.476,6.763,148.213
C01672=1225.127,292.472,-66.029,-176.474,6.766,148.213
C01673=1225.123,292.720,-66.059,-176.472,6.769,148.213
C01674=1225.118,292.969,-66.087,-176.470,6.771,148.213
C01675=1225.114,293.217,-66.116,-176.466,6.774,148.213
C01676=1225.110,293.466,-66.145,-176.464,6.776,148.213
C01677=1225.105,293.713,-66.174,-176.462,6.778,148.213
C01678=1225.101,293.961,-66.203,-176.460,6.780,148.212
C01679=1225.097,294.210,-66.232,-176.457,6.783,148.212
C01680=1225.092,294.459,-66.262,-176.455,6.785,148.212
C01681=1225.088,294.706,-66.290,-176.453,6.787,148.212
C01682=1225.084,294.955,-66.319,-176.450,6.790,148.212
C01683=1225.080,295.203,-66.348,-176.448,6.793,148.212
C01684=1225.075,295.451,-66.378,-176.445,6.795,148.212
C01685=1225.071,295.700,-66.406,-176.443,6.797,148.212
C01686=1225.066,295.948,-66.436,-176.441,6.800,148.212
C01687=1225.062,296.196,-66.465,-176.438,6.802,148.212
C01688=1225.058,296.445,-66.494,-176.436,6.804,148.211
C01689=1225.053,296.693,-66.523,-176.433,6.807,148.211
C01690=1225.050,296.941,-66.552,-176.431,6.809,148.211
C01691=1225.045,297.189,-66.581,-176.429,6.811,148.211
C01692=1225.041,297.437,-66.610,-176.426,6.814,148.211
C01693=1225.036,297.686,-66.639,-176.424,6.817,148.211
C01694=1225.032,297.934,-66.669,-176.422,6.819,148.211
C01695=1225.028,298.182,-66.698,-176.419,6.822,148.211
C01696=1225.023,298.430,-66.727,-176.417,6.824,148.211
C01697=1225.019,298.678,-66.757,-176.415,6.826,148.211
C01698=1225.015,298.927,-66.786,-176.413,6.828,148.211
C01699=1225.010,299.175,-66.815,-176.410,6.831,148.211
C01700=1225.006,299.424,-66.844,-176.407,6.833,148.210
C01701=1225.002,299.672,-66.874,-176.405,6.835,148.210
C01702=1224.998,299.920,-66.903,-176.403,6.839,148.210
C01703=1224.993,300.168,-66.932,-176.400,6.841,148.210
C01704=1224.989,300.416,-66.962,-176.398,6.843,148.210
C01705=1224.985,300.664,-66.991,-176.396,6.846,148.210
C01706=1224.981,300.912,-67.021,-176.394,6.848,148.210
C01707=1224.976,301.161,-67.050,-176.391,6.850,148.210
C01708=1224.972,301.410,-67.079,-176.388,6.853,148.210
C01709=1224.968,301.658,-67.108,-176.386,6.855,148.210
C01710=1224.964,301.906,-67.138,-176.384,6.858,148.210
C01711=1224.958,302.154,-67.168,-176.381,6.861,148.210
C01712=1224.954,302.402,-67.197,-176.379,6.863,148.210
C01713=1224.950,302.651,-67.226,-176.377,6.865,148.210
C01714=1224.945,302.899,-67.256,-176.375,6.868,148.210
C01715=1224.941,303.147,-67.285,-176.372,6.870,148.210
C01716=1224.937,303.395,-67.316,-176.370,6.873,148.209
C01717=1224.933,303.643,-67.345,-176.368,6.876,148.209
C01718=1224.929,303.891,-67.374,-176.365,6.878,148.209
C01719=1224.924,304.140,-67.405,-176.363,6.880,148.209
C01720=1224.920,304.388,-67.434,-176.360,6.883,148.209
C01721=1224.916,304.636,-67.463,-176.358,6.885,148.209
C01722=1224.912,304.885,-67.493,-176.356,6.887,148.209
C01723=1224.907,305.132,-67.522,-176.353,6.890,148.209
C01724=1224.903,305.380,-67.551,-176.351,6.892,148.209
C01725=1224.898,305.628,-67.582,-176.349,6.895,148.209
C01726=1224.894,305.877,-67.612,-176.347,6.898,148.209
C01727=1224.890,306.125,-67.641,-176.344,6.900,148.209
C01728=1224.885,306.373,-67.671,-176.342,6.902,148.209
C01729=1224.881,306.621,-67.700,-176.340,6.905,148.209
C01730=1224.876,306.870,-67.730,-176.338,6.907,148.209
C01731=1224.872,307.118,-67.760,-176.335,6.910,148.209
C01732=1224.868,307.366,-67.790,-176.333,6.913,148.209
C01733=1224.864,307.614,-67.819,-176.331,6.915,148.209
C01734=1224.859,307.863,-67.849,-176.329,6.917,148.209
C01735=1224.855,308.110,-67.879,-176.326,6.920,148.209
C01736=1224.851,308.359,-67.909,-176.324,6.922,148.209
C01737=1224.847,308.607,-67.938,-176.322,6.925,148.208
C01738=1224.842,308.855,-67.969,-176.319,6.928,148.208
C01739=1224.838,309.103,-67.998,-176.317,6.930,148.208
C01740=1224.834,309.351,-68.028,-176.315,6.932,148.208
C01741=1224.829,309.599,-68.059,-176.312,6.935,148.208
C01742=1224.825,309.848,-68.088,-176.310,6.937,148.208
C01743=1224.821,310.096,-68.118,-176.308,6.940,148.208
C01744=1224.816,310.344,-68.148,-176.305,6.943,148.208
C01745=1224.812,310.592,-68.178,-176.303,6.945,148.208
C01746=1224.808,310.840,-68.207,-176.301,6.947,148.208
C01747=1224.803,311.088,-68.238,-176.298,6.950,148.208
C01748=1224.800,311.337,-68.268,-176.296,6.952,148.208
C01749=1224.796,311.585,-68.298,-176.294,6.955,148.208
C01750=1224.791,311.834,-68.328,-176.292,6.958,148.208
C01751=1224.787,312.081,-68.358,-176.290,6.960,148.208
C01752=1224.782,312.330,-68.388,-176.287,6.963,148.208
C01753=1224.778,312.578,-68.418,-176.285,6.965,148.208
C01754=1224.774,312.826,-68.448,-176.283,6.968,148.208
C01755=1224.769,313.074,-68.478,-176.280,6.971,148.208
C01756=1224.765,313.322,-68.508,-176.278,6.973,148.208
C01757=1224.760,313.571,-68.538,-176.276,6.975,148.208
C01758=1224.757,313.818,-68.568,-176.274,6.978,148.208
C01759=1224.753,314.066,-68.598,-176.271,6.980,148.208
C01760=1224.748,314.315,-68.629,-176.270,6.983,148.208
C01761=1224.745,314.563,-68.659,-176.267,6.986,148.208
C01762=1224.740,314.811,-68.689,-176.265,6.988,148.208
C01763=1224.736,315.087,-68.723,-176.262,6.991,148.208
C01764=1224.730,315.363,-68.756,-176.260,6.994,148.208
C01765=1224.725,315.638,-68.790,-176.258,6.997,148.208
C01766=1224.721,315.914,-68.823,-176.255,7.000,148.208
C01767=1224.716,316.162,-68.854,-176.253,7.002,148.208
C01768=1224.712,316.410,-68.884,-176.250,7.005,148.208
C01769=1224.707,316.659,-68.914,-176.248,7.007,148.208
C01770=1224.704,316.907,-68.945,-176.246,7.011,148.208
C01771=1224.699,317.155,-68.976,-176.244,7.013,148.208
C01772=1224.695,317.403,-69.005,-176.242,7.015,148.208
C01773=1224.691,317.651,-69.036,-176.239,7.018,148.208
C01774=1224.687,317.899,-69.066,-176.237,7.020,148.208
C01775=1224.682,318.147,-69.096,-176.235,7.023,148.208
C01776=1224.679,318.396,-69.126,-176.233,7.026,148.208
C01777=1224.674,318.644,-69.157,-176.231,7.028,148.208
C01778=1224.669,318.892,-69.188,-176.228,7.030,148.208
C01779=1224.666,319.139,-69.218,-176.226,7.033,148.208
C01780=1224.661,319.388,-69.248,-176.224,7.036,148.208
C01781=1224.657,319.636,-69.279,-176.222,7.039,148.208
C01782=1224.653,319.884,-69.310,-176.219,7.041,148.208
C01783=1224.648,320.132,-69.340,-176.217,7.043,148.208
C01784=1224.644,320.380,-69.370,-176.215,7.047,148.208
C01785=1224.639,320.628,-69.401,-176.213,7.049,148.208
C01786=1224.636,320.877,-69.431,-176.211,7.051,148.208
C01787=1224.631,321.125,-69.462,-176.208,7.054,148.208
C01788=1224.627,321.373,-69.493,-176.207,7.057,148.208
C01789=1224.623,321.620,-69.523,-176.204,7.060,148.208
C01790=1224.619,321.869,-69.554,-176.202,7.062,148.208
C01791=1224.614,322.117,-69.585,-176.200,7.065,148.209
C01792=1224.610,322.365,-69.615,-176.198,7.068,148.209
C01793=1224.606,322.612,-69.646,-176.195,7.070,148.209
C01794=1224.602,322.861,-69.677,-176.193,7.072,148.209
C01795=1224.598,323.109,-69.707,-176.191,7.075,148.209
C01796=1224.593,323.357,-69.738,-176.189,7.078,148.209
C01797=1224.589,323.605,-69.769,-176.187,7.080,148.209
C01798=1224.585,323.853,-69.800,-176.185,7.083,148.209
C01799=1224.581,324.101,-69.830,-176.183,7.085,148.209
C01800=1224.576,324.349,-69.860,-176.180,7.088,148.209
C01801=1224.572,324.598,-69.892,-176.178,7.091,148.209
C01802=1224.568,324.846,-69.922,-176.176,7.093,148.209
C01803=1224.564,325.093,-69.953,-176.174,7.096,148.209
C01804=1224.560,325.342,-69.984,-176.172,7.099,148.209
C01805=1224.555,325.590,-70.014,-176.170,7.101,148.209
C01806=1224.550,325.838,-70.045,-176.168,7.104,148.209
C01807=1224.547,326.086,-70.076,-176.166,7.107,148.209
C01808=1224.543,326.334,-70.106,-176.163,7.110,148.209
C01809=1224.538,326.582,-70.137,-176.161,7.112,148.209
C01810=1224.534,326.831,-70.168,-176.159,7.114,148.209
C01811=1224.529,327.079,-70.199,-176.157,7.118,148.210
C01812=1224.526,327.326,-70.230,-176.155,7.120,148.210
C01813=1224.522,327.574,-70.261,-176.153,7.122,148.210
C01814=1224.517,327.822,-70.292,-176.151,7.126,148.210
C01815=1224.513,328.070,-70.323,-176.149,7.128,148.210
C01816=1224.509,328.319,-70.354,-176.147,7.130,148.210
C01817=1224.504,328.566,-70.385,-176.144,7.133,148.210
C01818=1224.500,328.814,-70.416,-176.143,7.136,148.210
C01819=1224.496,329.063,-70.447,-176.140,7.139,148.210
C01820=1224.492,329.311,-70.477,-176.138,7.141,148.210
C01821=1224.488,329.559,-70.509,-176.136,7.144,148.210
